IF (lCurrentTime.Value > (lToggleTime + lTogglePeriodMicroseconds)) THEN
	lToggle := NOT(lToggle);
	lToggleTime := lCurrentTime.Value;
END_IF

IF (lCurrentTime.Value > lIntegralClockTickPrevious) THEN
	lIntegralClockTick := TRUE;
	lIntegralClockTickPrevious := lIntegralClockTickPrevious + lIntegralPeriod;
ELSE
	lIntegralClockTick := FALSE;
END_IF

IF (lIntegralRunning) THEN
	lIntegralDuration := lCurrentTime.Value - lIntegralStartTime;
ELSE
	lIntegralStartTime := lCurrentTime.Value;
END_IF
IF (lIntegralReset) THEN
	lIntegralDuration := 0;
	lIntegralReset := FALSE;
END_IF

lCounter := lCounter + 1;


                
END_METHOD

METHOD initializeCycle
  VAR_INPUT
    currentTime : REFERENCE TO ULINT;
  END_VAR
                  lCurrentTime.InputReference REF= currentTime;

                
END_METHOD

METHOD describe
  VAR_INPUT
    executeContext : POINTER TO ExecuteContext;
  END_VAR
                  SUPER^.describe(executeContext);

IF (executeContext^.matchOption(cExecuteOptionSyntax)) THEN
	RETURN;
END_IF

IF (executeContext^.matchOption(cExecuteOptionParameter)) THEN	
	RETURN;
END_IF

executeContext^.appendPair('current_time',TIME_TO_STRING(ULINT_TO_TIME(lCurrentTime.Value/1000)),TRUE,TRUE);
executeContext^.appendPair('start_time',TIME_TO_STRING(ULINT_TO_TIME(lStartTime.Value/1000)),TRUE,TRUE);
executeContext^.appendPair('up_time',TIME_TO_STRING(ULINT_TO_TIME((lCurrentTime.Value - lStartTime.Value)/1000)),TRUE,TRUE);
executeContext^.appendPair('system_time',SystemTime,TRUE,TRUE);
executeContext^.appendPair('time_step',gTypeHandler.getTokenForUDINT(lTimeStep),FALSE,TRUE);

                
END_METHOD

METHOD configure
  VAR_INPUT
    executeContext : POINTER TO ExecuteContext;
  END_VAR
  VAR
    b : BOOL;
  END_VAR
                  IF (gSystemServices.Initialized) THEN
	IF (executeContext^.configureBool(cTokenFailSafeConfig,b,FALSE,0)) THEN
		RETURN;
	END_IF
END_IF

SUPER^.configure(executeContext);

                
END_METHOD

PROPERTY AverageCycleTime : ULINT
GET
                    AverageCycleTime := lAverageCycleTime;

                  
END_GET
END_PROPERTY

PROPERTY CycleTime : ULINT
GET
                    CycleTime := lCycleTime;

                  
END_GET
END_PROPERTY

PROPERTY Hours : REAL
GET
                    Hours := 0;
                  
END_GET
SET
                    
                  
END_SET
END_PROPERTY

PROPERTY IntegralClockTick : BOOL
GET
                    IntegralClockTick := lIntegralClockTick;
                  
END_GET
END_PROPERTY

PROPERTY OperationalHours : REAL
GET
                    OperationalHours := 0;
                  
END_GET
SET
                    
                  
END_SET
END_PROPERTY

PROPERTY SystemTime : REFERENCE TO t_medium_string
GET
                    SystemTime REF= lSystemTime;

                  
END_GET
END_PROPERTY

PROPERTY TimeStep : t_timestep
GET
                    TimeStep := lTimeStep;
                  
END_GET
END_PROPERTY

PROPERTY Toggle : BOOL
GET
                    Toggle := lToggle;
                  
END_GET
END_PROPERTY

PROPERTY TypeToken : t_medium_string
GET
                    TypeToken := 'Cycle';
                  
END_GET
END_PROPERTY

PROPERTY SystemTimeMicroseconds : ULINT
GET
                    SystemTimeMicroseconds := lCurrentTime.Value;
                  
END_GET
END_PROPERTY

PROPERTY StartCount : UINT
GET
                    StartCount := lStartCount.Value;
                  
END_GET
END_PROPERTY

PROPERTY StartTimeMicroseconds : ULINT
GET
                    StartTimeMicroseconds := 0; //lStartTime.Value;
                  
END_GET
END_PROPERTY
END_FUNCTION_BLOCK

FUNCTION_BLOCK Executor EXTENDS OperationalParticleSet
  VAR CONSTANT
    cCommandQueueMax : USINT := 4;
  END_VAR
  VAR
    lAlarmSoftwareCrash : ReportableAlarm;
    lClient : TCPClient;
    lExecuteContext : ExecuteContextExecutor;
    lExecuteContextParameterUpdate : ExecuteContextExecutor;
    lEnabled : BOOL := TRUE;
    lCommandQueue : ARRAY[1..cCommandQueueMax] OF t_command_request;
    lQueueCount : USINT := 0;
  END_VAR

            
          

METHOD operator
  VAR
    length : UINT;
  END_VAR
                  SUPER^.operator();

lExecuteContext.operator();
IF (lEnabled) THEN
	lClient.write(lExecuteContext.WriteStream^.Buffer,lExecuteContext.WriteStream^.Characters);
	lClient.write(lExecuteContextParameterUpdate.WriteStream^.Buffer,lExecuteContextParameterUpdate.WriteStream^.Characters);
END_IF

lExecuteContextParameterUpdate.WriteStream^.clear();

                
END_METHOD

METHOD initialize
                  lExecuteContext.Source REF= THIS^;
// lExecuteContextParameterUpdate.Source REF= THIS^; dummy executor: provides context only for direct write out

lAlarmSoftwareCrash.initializeState(NopSelf,'',cACExecutionFailed);

registerOperational(ADR(lClient));

SUPER^.initialize();

lExecuteContext.WriteStream^.IndentStr := '';
lExecuteContext.WriteStream^.NewlineStr := '$n';
lExecuteContext.WriteStream^.RecordInitiatorStr := '{';
lExecuteContext.WriteStream^.RecordTerminatorStr := '}';
lExecuteContext.WriteStream^.clear();
lExecuteContext.EnableExecutor := FALSE;

lExecuteContextParameterUpdate.WriteStream^.IndentStr := '';
lExecuteContextParameterUpdate.WriteStream^.NewlineStr := '$n';
lExecuteContextParameterUpdate.WriteStream^.RecordInitiatorStr := '{';
lExecuteContextParameterUpdate.WriteStream^.RecordTerminatorStr := '}';
lExecuteContextParameterUpdate.WriteStream^.clear();
lExecuteContextParameterUpdate.Command.optionCount := 1;
lExecuteContextParameterUpdate.Command.options[1] := cExecuteOptionParameter;
lExecuteContextParameterUpdate.EnableExecutor := FALSE;

                
END_METHOD

METHOD getNextExecuteCommand : BOOL
  VAR_INPUT
    command : REFERENCE TO t_command_request;
  END_VAR
  VAR
    i : USINT;
  END_VAR
                  IF (lQueueCount=0) THEN
	getNextExecuteCommand := FALSE;
	RETURN;
END_IF

command := lCommandQueue[1];

FOR i:=1 TO lQueueCount-1 DO
	lCommandQueue[i] := lCommandQueue[i+1];
END_FOR

lQueueCount := lQueueCount - 1;

getNextExecuteCommand := TRUE;

                
END_METHOD

METHOD reportParameterUpdates
  VAR_INPUT
    particle : POINTER TO t_particle;
  END_VAR
                  IF (particle=0) THEN
	RETURN;
END_IF

particle^.describe(ADR(lExecuteContextParameterUpdate));

                
END_METHOD

METHOD putCommand : BOOL
  VAR_INPUT
    command : REFERENCE TO t_command_request;
  END_VAR
                  IF (lQueueCount=cCommandQueueMax) THEN
	putCommand := FALSE;
	RETURN;
END_IF

lQueueCount := lQueueCount + 1;
lCommandQueue[lQueueCount] := command;

putCommand := TRUE;

                
END_METHOD

PROPERTY Client : REFERENCE TO TCPClient
GET
                    Client ref= lClient;
                  
END_GET
END_PROPERTY

PROPERTY TypeToken : t_medium_string
GET
                    TypeToken := 'Executor';
                  
END_GET
END_PROPERTY

PROPERTY ExecuteContext : POINTER TO ExecuteContextExecutor
GET
                    ExecuteContext:= ADR(lExecuteContext);
                  
END_GET
END_PROPERTY
END_FUNCTION_BLOCK

FUNCTION fCheckChannelMask : BOOL
  VAR_INPUT
    set : UINT;
    mask : t_channel_mask;
  END_VAR

            fCheckChannelMask := UINT_TO_BOOL(set AND INT_TO_UINT(mask));

          
END_FUNCTION

FUNCTION fCheckDebugFlags : BOOL
  VAR_INPUT
    mask : t_debug_mask;
  END_VAR

            fCheckDebugFlags := UINT_TO_BOOL(gDebugFlags.Value AND INT_TO_UINT(mask));

          
END_FUNCTION

FUNCTION_BLOCK LEDDiagnostic EXTENDS OperationalParticleSet
  VAR
    lCode : t_led_code;
  END_VAR

            
          

METHOD initialize
                  SUPER^.initialize();
SubSystem := cSubsystemPowerpack;

                
END_METHOD

METHOD operator
  VAR
    i : USINT;
  END_VAR
                  SUPER^.operator();

lCode := cLEDCodeNone;

                
END_METHOD

METHOD configure
  VAR_INPUT
    executeContext : POINTER TO ExecuteContext;
  END_VAR
  VAR
    b : BOOL;
  END_VAR
                  IF (gSystemServices.Initialized) THEN
	IF (executeContext^.configureBool(cTokenFailSafeConfig,b,FALSE,0)) THEN
		RETURN;
	END_IF
END_IF

SUPER^.configure(executeContext);

                
END_METHOD

PROPERTY TypeToken : t_medium_string
GET
                    TypeToken := 'LED';
                  
END_GET
END_PROPERTY

PROPERTY Code : t_led_code
GET
                    Code := lCode;
                  
END_GET
SET
                    // exceptions to the order rule
lCode := MAX(Code,lCode);

                  
END_SET
END_PROPERTY
END_FUNCTION_BLOCK

FUNCTION_BLOCK LocalMachine EXTENDS NonOperationalParticleSet
  VAR CONSTANT
    cRecoveryDetectionSteps : USINT := 3;
    cRecoverDetectionInterval : t_time := TIME#1s0ms;
  END_VAR
  VAR
    lVRMachineName : ValueReferencePersistentMediumString;
    lMachineName : t_persistent_medium_string;
    lVRDebugFlags : ValueReferencePersistentUINT;
    lVRFailSafeDebugFlags : ValueReferencePersistentUINT;
    lFailSafeDebugFlags : t_persistent_uint;
    lRecoveryDetectionStep : t_persistent_uint;
    lRecoveryDetectionStepActive : t_persistent_bool;
    lRecoveryDetectionPeriods : ARRAY[0..cRecoveryDetectionSteps] OF t_time;
    lRecoveryDetectionTimerLower : t_timer;
    lRecoveryDetectionTimerUpper : t_timer;
    lRecoveryDetectionSuccess : BOOL := FALSE;
    lPostInitialize : BOOL := TRUE;
  END_VAR

            
          

METHOD execute
  VAR_INPUT
    executeContext : POINTER TO ExecuteContext;
  END_VAR
  VAR
    token : t_token_string;
    mask : t_debug_mask;
  END_VAR
                  IF (executeContext=0) THEN
	RETURN;
END_IF

IF (executeContext^.matchCommand(sCommandDebugMaskAdd)) THEN

	IF (NOT(executeContext^.configureEnum(cEnumTypeDebugMask,cTokenFeature,mask,TRUE,THIS))) THEN
		RETURN;
	END_IF
	
	gDebugFlags.Value := gDebugFlags.Value OR INT_TO_UINT(mask);
	RETURN;
END_IF

IF (executeContext^.matchCommand(sCommandDebugMaskDelete)) THEN

	IF (NOT(executeContext^.configureEnum(cEnumTypeDebugMask,cTokenFeature,mask,TRUE,THIS))) THEN
		RETURN;
	END_IF
	
	gDebugFlags.Value := gDebugFlags.Value AND NOT(INT_TO_UINT(mask));
	RETURN;
END_IF

IF (executeContext^.matchCommand(sCommandDebugMaskClear)) THEN	
	gDebugFlags.Value := 0;
	RETURN;
END_IF

SUPER^.execute(executeContext);

                
END_METHOD

METHOD postInitialize
                  lPostInitialize := false;
                
END_METHOD

METHOD initialize
                  lVRDebugFlags.initializeValueReference(gDebugFlags,NopSelf,'Debug','System wide debug flags','',cValueStyleParameter);

lVRFailSafeDebugFlags.initializeValueReference(lFailSafeDebugFlags,NopSelf,'FailSafeDebug','Failsafe debug flags','',cValueStyleParameter);
lFailSafeDebugFlags.Identifier := t_persistent_id.cPersistentID_FailSafeDebugFlags;
lFailSafeDebugFlags.initialize();

lVRMachineName.initializeValueReference(lMachineName,NopSelf,'MachineName','Name of the machine','',cValueStyleParameter);
lMachineName.Identifier := t_persistent_id.cPersistentID_MachineName;
lMachineName.initialize();

lRecoveryDetectionStep.Identifier := t_persistent_id.cPersistentID_RecoveryDetectionStep;
lRecoveryDetectionStep.initialize();

lRecoveryDetectionStepActive.Identifier := t_persistent_id.cPersistentID_RecoveryDetectionStepActive;
lRecoveryDetectionStepActive.initialize();

SUPER^.initialize();
SubSystem := cSubsystemMachine;

lRecoveryDetectionPeriods[0] := T#500MS;
lRecoveryDetectionPeriods[1] := T#2500MS;
lRecoveryDetectionPeriods[2] := T#500MS;
lRecoveryDetectionPeriods[3] := T#2500MS;

lRecoveryDetectionTimerLower.Enable := TRUE;
lRecoveryDetectionTimerLower.Period := lRecoveryDetectionPeriods[MIN(lRecoveryDetectionStep.Value,cRecoveryDetectionSteps)];
lRecoveryDetectionTimerLower.initialize();

lRecoveryDetectionTimerUpper.Enable := TRUE;
lRecoveryDetectionTimerUpper.Period := lRecoveryDetectionPeriods[MIN(lRecoveryDetectionStep.Value,cRecoveryDetectionSteps)] + cRecoverDetectionInterval;
lRecoveryDetectionTimerUpper.initialize();

IF (lRecoveryDetectionStepActive.Value) THEN
	lRecoveryDetectionStep.Value := lRecoveryDetectionStep.Value + 1;
	lRecoveryDetectionStepActive.Value := FALSE;
END_IF

IF (lRecoveryDetectionStep.Value>cRecoveryDetectionSteps) THEN
	lRecoveryDetectionStep.Value := 0;
	lRecoveryDetectionSuccess := TRUE;
	gDebugFlags.Value := INT_TO_UINT(cDebugDisableWatchdog);
END_IF
                
END_METHOD

METHOD operator
                  SUPER^.operator();

IF (gSystemServices.PLC.CrashSeverity>3) THEN
	lFailSafeDebugFlags.Value := INT_TO_UINT(cDebugDisableWatchdog);
END_IF

IF (gSystemServices.PLC.CrashSeverity>2) THEN
	gDebugFlags.Value := lFailSafeDebugFlags.Value;
END_IF

IF (lRecoveryDetectionTimerUpper.Enable) THEN
	lRecoveryDetectionTimerLower.operator();
	lRecoveryDetectionTimerUpper.operator();

	lRecoveryDetectionStepActive.Value := ((lRecoveryDetectionTimerLower.Expired) AND
		(NOT(lRecoveryDetectionTimerUpper.Expired)));

	IF ((lRecoveryDetectionTimerLower.Expired) AND
		(lRecoveryDetectionTimerUpper.Expired)) THEN
		lRecoveryDetectionTimerLower.Enable := FALSE;
		lRecoveryDetectionTimerUpper.Enable := FALSE;
		lRecoveryDetectionStep.Value := 0;
	END_IF
END_IF

IF (lPostInitialize) THEN
	postInitialize();
END_IF

                
END_METHOD

METHOD defaultPersistence
                  lFailSafeDebugFlags.Value := INT_TO_UINT(cDebugDisableWatchdog);
                
END_METHOD

METHOD describe
  VAR_INPUT
    executeContext : POINTER TO ExecuteContext;
  END_VAR
                  SUPER^.describe(executeContext);

IF (executeContext^.matchOption(cExecuteOptionSyntax)) THEN
	executeContext^.describeSyntaxExecutable(sCommandDebugMaskAdd);
	executeContext^.describeSyntaxExecutable(sCommandDebugMaskDelete);
	executeContext^.describeSyntaxExecutable(sCommandDebugMaskClear);

	RETURN;
END_IF

IF (executeContext^.matchOption(cExecuteOptionParameter)) THEN	
	RETURN;
END_IF

executeContext^.appendPair('machine_name',lMachineName.Value,TRUE,TRUE);


                
END_METHOD

METHOD configure
  VAR_INPUT
    executeContext : POINTER TO ExecuteContext;
  END_VAR
  VAR
    b : BOOL;
  END_VAR
                  IF (gSystemServices.Initialized) THEN
	IF (executeContext^.configureBool(cTokenFailSafeConfig,b,FALSE,0)) THEN
		RETURN;
	END_IF
END_IF

SUPER^.configure(executeContext);

                
END_METHOD

PROPERTY MachineName : t_medium_string
GET
                    MachineName := lMachineName.Value;
                  
END_GET
SET
                    lMachineName.Value := MachineName;
                  
END_SET
END_PROPERTY

PROPERTY TypeToken : t_medium_string
GET
                    TypeToken := 'Local';
                  
END_GET
END_PROPERTY
END_FUNCTION_BLOCK

FUNCTION_BLOCK Peripheral EXTENDS OperationalParticleSet
  VAR
    lExternalState : REFERENCE TO UINT;
    lSupplementaryCommand : REFERENCE TO USINT;
    lInternalState : REFERENCE TO USINT;
    lReportableState : REFERENCE TO UDINT;
    lSupplementaryState : REFERENCE TO UINT;
    lOperatingModeLockRequest : ValueObjectBoolInputReferenceUSINT;
    lOperatingModeRunningRegister : ValueObjectBoolInputReferenceUSINT;
    lUMFSRegister : ValueObjectBoolInputReferenceUSINT;
    lValidTransmissions : ValueObjectBoolInputReferenceUSINT;
    lTPDO1Stuffing : ValueObjectBoolInputReferenceUSINT;
    lReportable : ARRAY[0..31] OF POINTER TO t_reportable;
  END_VAR

            ;
          

METHOD initialize
                  IF ((NOT(__ISVALIDREF(lExternalState))) OR
	(NOT(__ISVALIDREF(lSupplementaryCommand))) OR
	(NOT(__ISVALIDREF(lInternalState))) OR
	(NOT(__ISVALIDREF(lReportableState))) OR
	(NOT(__ISVALIDREF(lSupplementaryState)))) THEN
	gCodeErrorHandler(pMessage:=CONCAT('null reference in ',lIdentity));
END_IF

lOperatingModeLockRequest.initializeValueObjectOp(OpSelf,'LockReq','Lock operating mode requested','',cValueStyleConfigurable);
lOperatingModeLockRequest.Index := 0;
lOperatingModeLockRequest.InputReference REF= lInternalState;

lOperatingModeRunningRegister.initializeValueObjectOp(OpSelf,'RunningReg','Running operating mode requested','',cValueStyleConfigurable);
lOperatingModeRunningRegister.Index := 1;
lOperatingModeRunningRegister.InputReference REF= lInternalState;

lUMFSRegister.initializeValueObjectOp(OpSelf,'UMFSReg','UMFS registration requested','',cValueStyleConfigurable);
lUMFSRegister.Index := 2;
lUMFSRegister.InputReference REF= lInternalState;

lValidTransmissions.initializeValueObjectOp(OpSelf,'ValidTrnsmssns','Valid transmissions detected','',cValueStyleConfigurable);
lValidTransmissions.Index := 3;
lValidTransmissions.InputReference REF= lInternalState;

lTPDO1Stuffing.initializeValueObjectOp(OpSelf,'TPDO1Stuffing','TPDO1 stuffing bit detected','',cValueStyleConfigurable);
lTPDO1Stuffing.Index := 7;
lTPDO1Stuffing.InputReference REF= lInternalState;

SUPER^.initialize();
                
END_METHOD

METHOD initializePeripheral
  VAR_INPUT
    externalState : REFERENCE TO UINT;
    supplementaryCommand : REFERENCE TO USINT;
    internalState : REFERENCE TO USINT;
    reportableState : REFERENCE TO UDINT;
    supplementaryState : REFERENCE TO UINT;
  END_VAR
                  lExternalState REF= externalState;
lSupplementaryCommand REF= supplementaryCommand;

lInternalState REF= internalState;
lReportableState REF= reportableState;
lSupplementaryState REF= supplementaryState;



                
END_METHOD

METHOD operator
  VAR
    i : USINT;
    u : UDINT;
  END_VAR
                  SUPER^.operator();

(* traffic FROM master PLC *)

lExternalState := 0;
lExternalState := fMergeBoolIntoWord(pWord:=lExternalState,pData:=gManualTemporaryOveride,pStart:=9);

(* traffic to master PLC *)

u := lReportableState;
FOR i:=0 TO 15 DO
	IF ((UDINT_TO_BOOL(u AND 2#1)) AND
		(lReportable[i]<>0)) THEN
		lReportable[i]^.trigger(FALSE);
	END_IF
	
	u := SHR(u,1);
END_FOR

                
END_METHOD

METHOD registerReportable
  VAR_INPUT
    reportable : POINTER TO t_reportable;
    index : USINT;
  END_VAR
                  IF (index>31) THEN
	RETURN;
END_IF

lReportable[index] := reportable;

                
END_METHOD

PROPERTY TPDO1Stuffing : BOOL
GET
                    TPDO1Stuffing := lTPDO1Stuffing.Value;
                  
END_GET
END_PROPERTY

PROPERTY TypeToken : t_medium_string
GET
                    TypeToken := 'Peripheral';
                  
END_GET
END_PROPERTY

PROPERTY ValidTransmissions : BOOL
GET
                    ValidTransmissions := lValidTransmissions.Value;
                  
END_GET
END_PROPERTY

PROPERTY SupplementaryCommand : REFERENCE TO USINT
GET
                    SupplementaryCommand ref= lSupplementaryCommand;
                  
END_GET
END_PROPERTY

PROPERTY SupplementaryState : REFERENCE TO UINT
GET
                    SupplementaryState ref= lSupplementaryState;
                  
END_GET
END_PROPERTY
END_FUNCTION_BLOCK

FUNCTION_BLOCK PLC EXTENDS OperationalParticleSet
  VAR CONSTANT
    cCrashDetectionPeriod : t_time := TIME#30s0ms;
    cPersistedCommandCount : USINT := 100;
  END_VAR
  VAR
    lVRTriggerWipePersistence : ValueReferenceBool;
    lTriggerWipePersistence : BOOL := FALSE;
    lVRTriggerDefaultPersistence : ValueReferenceBool;
    lTriggerDefaultPersistence : BOOL := FALSE;
    lVRTriggerResetSoftwareCrashCount : ValueReferenceBool;
    lTriggerResetSoftwareCrashCount : BOOL := FALSE;
    lVRTemporaryDisableWatchdog : ValueReferencePersistentBool;
    lTemporaryDisableWatchdog : t_persistent_bool;
    lVRMaintenanceMode : ValueReferenceBool;
    lMaintenanceMode : BOOL := FALSE;
    lMaintenanceModePrevious : BOOL := FALSE;
    lAlarmSoftwareCrash : ReportableAlarm;
    lAlarmFailSafeMode : ReportableAlarm;
    lAlarmMaintenanceMode : ReportableAlarm;
    lAlarmWatchdogDisabled : ReportableAlarm;
    lAlarmPersistedCommands : ReportableAlarm;
    lShutdownCode : t_persistent_int;
    lPreviousShutdownCode : t_shutdown_code;
    lSoftwareCrashCount : t_persistent_uint;
    lCrashSeverity : t_persistent_uint;
    lCrashDetectionTimer : t_timer;
    lCrashDetected : BOOL := FALSE;
    lTrapDetected : BOOL := FALSE;
    lFailSafeModeActive : BOOL := FALSE;
    lDisableWatchDog : BOOL := FALSE;
    lForceDisableWatchDog : BOOL := FALSE;
    lPersistedCommands : ARRAY[1..cPersistedCommandCount] OF PersistentCommand;
    lPersistedCommandCount : UINT;
    lPersistedCommandsStatus : BOOL := TRUE;
  END_VAR

            
          

METHOD setFailSafeMode
                  lFailSafeModeActive := TRUE;

setWatchdog();


                
END_METHOD

METHOD clearFailSafeMode
                  lFailSafeModeActive := FALSE;

setWatchdog();

                
END_METHOD

METHOD operator
  VAR
    i : USINT;
  END_VAR
                  SUPER^.operator();

IF (lTriggerWipePersistence) THEN
	lTriggerWipePersistence := FALSE;

	gPersistenceManager.clear();

	defaultPersistence();
	gSystemServices.LocalMachine.defaultPersistence();
END_IF

IF (lTriggerDefaultPersistence) THEN
	lTriggerDefaultPersistence := FALSE;

	defaultPersistence();
	gSystemServices.LocalMachine.defaultPersistence();
END_IF
	
IF (lTriggerResetSoftwareCrashCount) THEN
	lTriggerResetSoftwareCrashCount := FALSE;

	lSoftwareCrashCount.Value := 0;
END_IF

IF (lCrashDetectionTimer.Enable) THEN
	lCrashDetectionTimer.operator();
	IF (lCrashDetectionTimer.Expired) THEN
		lCrashDetectionTimer.Enable := FALSE;
		lShutdownCode.Value := t_shutdown_code.cShutdownCodeUnknown;
	END_IF
END_IF

IF ((lCrashDetected) OR (lTrapDetected)) THEN
	lAlarmSoftwareCrash.trigger(FALSE);
	gSystemServices.LEDDiagnostic.Code := cLEDCodeSoftwareCrash;
END_IF

IF (lFailSafeModeActive) THEN
	lAlarmFailSafeMode.trigger(FALSE);

	IF (lCrashSeverity.Value>1) THEN
		gSystemServices.LEDDiagnostic.Code := cLEDCodeFailSafeSevere;			
	ELSE
		gSystemServices.LEDDiagnostic.Code := cLEDCodeFailSafe;
	END_IF
END_IF

IF (MaintenanceMode<>lMaintenanceModePrevious) THEN
	lMaintenanceModePrevious := MaintenanceMode;
	setWatchdog();	
END_IF

IF (MaintenanceMode)  THEN
	lAlarmMaintenanceMode.trigger(FALSE);
	gSystemServices.LEDDiagnostic.Code := cLEDCodeMaintenance;
END_IF

IF (fCheckDebugFlags(cDebugDisableWatchdog)<>lDisableWatchDog) THEN
	lDisableWatchDog := NOT(lDisableWatchDog);
	setWatchdog();
END_IF

IF ((lDisableWatchDog) OR (lForceDisableWatchDog)) THEN
	lAlarmWatchdogDisabled.trigger(FALSE);
	gSystemServices.LEDDiagnostic.Code := cLEDCodeWatchDogDisabled;	
END_IF

IF (NOT(lPersistedCommandsStatus)) THEN
	lAlarmPersistedCommands.trigger(FALSE);
END_IF

                
END_METHOD

METHOD initialize
  VAR
    i : USINT;
    id : INT;
  END_VAR
                  lVRTriggerWipePersistence.initializeValueReference(lTriggerWipePersistence,NopSelf,'WipePersist','Trigger wipe of persistent memory','',cValueStyleTrigger);
lVRTriggerDefaultPersistence.initializeValueReference(lTriggerDefaultPersistence,NopSelf,'DefaultPersist','Trigger loading default persistent memory','',cValueStyleTrigger);
lVRTriggerResetSoftwareCrashCount.initializeValueReference(lTriggerResetSoftwareCrashCount,NopSelf,'ResetOpSwCrshCnt','Trigger reset software crash count','',cValueStyleTrigger);
lVRMaintenanceMode.initializeValueReference(lMaintenanceMode,NopSelf,'Maintenance','Whether in maintenance mode','',cValueStyleParameter);

lVRTemporaryDisableWatchdog.initializeValueReference(lTemporaryDisableWatchdog,NopSelf,'TmpDsblWatchDog','Temporarily disable watchdog','',cValueStyleParameter);
lTemporaryDisableWatchdog.Identifier := t_persistent_id.cPersistentID_TemporaryDisableWatchdog;
lTemporaryDisableWatchdog.initialize();

lAlarmSoftwareCrash.initializeState(NopSelf,'',cACSoftwareCrash);
lAlarmFailSafeMode.initializeState(NopSelf,'',cACFailSafeMode);
lAlarmMaintenanceMode.initializeState(NopSelf,'',cACMaintenanceMode);
lAlarmWatchdogDisabled.initializeState(NopSelf,'',cACWatchdogDisabled);
lAlarmPersistedCommands.initializeState(NopSelf,'',cACPersistedCommands);

lShutdownCode.Identifier := t_persistent_id.cPersistentID_ShutdownCode;
lShutdownCode.initialize();

lSoftwareCrashCount.Identifier := t_persistent_id.cPersistentID_SoftwareCrashCount;
lSoftwareCrashCount.initialize();

lCrashSeverity.Identifier := t_persistent_id.cPersistentID_CrashSeverity;
lCrashSeverity.initialize();

lDisableWatchDog := fCheckDebugFlags(cDebugDisableWatchdog);

IF (lTemporaryDisableWatchdog.Value) THEN
	lTemporaryDisableWatchdog.Value := FALSE;	
	lForceDisableWatchDog := TRUE;
END_IF

lPersistedCommandCount := 0;
id := t_persistent_id.cPersistentID_CommandRepositoryLower;

FOR i:=1 TO cPersistedCommandCount DO
	lPersistedCommands[i].Identifier := id;
	lPersistedCommands[i].initialize();
	
	id := id + UINT_TO_INT(lPersistedCommands[i].Blocks);
	
	IF (lPersistedCommands[i].Valid) THEN
		lPersistedCommandCount := lPersistedCommandCount + 1;
	END_IF
END_FOR
	
SUPER^.initialize();

lPreviousShutdownCode := lShutdownCode.Value;
lShutdownCode.Value := t_shutdown_code.cShutdownCodeCrashDetected;

lCrashDetected := (lPreviousShutdownCode=t_shutdown_code.cShutdownCodeCrashDetected);
IF (lCrashDetected) THEN		
	lCrashSeverity.Value := lCrashSeverity.Value + 1;
	lSoftwareCrashCount.Value := lSoftwareCrashCount.Value + 1;
ELSE
	lCrashSeverity.Value := 0;
END_IF

lCrashDetectionTimer.Enable := TRUE;
lCrashDetectionTimer.Period := cCrashDetectionPeriod;
lCrashDetectionTimer.initialize();

                
END_METHOD

METHOD describe
  VAR_INPUT
    executeContext : POINTER TO ExecuteContext;
  END_VAR
  VAR
    i : UINT;
    str : STRING;
    store : t_command_store;
    particle : t_particle_ptr;
    token : t_token_string;
  END_VAR
                  SUPER^.describe(executeContext);

IF (executeContext^.matchOption(cExecuteOptionSyntax)) THEN
	executeContext^.describeSyntaxExecutable(sCommandExport);
	executeContext^.describeSyntaxExecutable(sCommandClear);
	executeContext^.describeSyntaxExecutable(sCommandExecute);

	RETURN;
END_IF

IF (executeContext^.matchOption(cExecuteOptionParameter)) THEN	
	RETURN;
END_IF

executeContext^.appendPair('failsafe_active',gTypeHandler.getTokenForBool(lFailSafeModeActive),FALSE,TRUE);
executeContext^.appendPair('crash_detected',gTypeHandler.getTokenForBool(lCrashDetected),FALSE,TRUE);
executeContext^.appendPair('crash_severity',gTypeHandler.getTokenForUINT(lCrashSeverity.Value),FALSE,TRUE);
executeContext^.appendPair('previous_shutdown',gTypeHandler.getTokenForEnum(cEnumTypeShutdownCode,lPreviousShutdownCode),TRUE,TRUE);
executeContext^.appendPair('watchdog',gTypeHandler.getTokenForBool(NOT((lDisableWatchdog) OR (lForceDisableWatchDog))),FALSE,TRUE);
executeContext^.appendPair('persisted_count',gTypeHandler.getTokenForUINT(lPersistedCommandCount),FALSE,TRUE);
executeContext^.appendPair('persisted_status',gTypeHandler.getTokenForBool(lPersistedCommandsStatus),FALSE,TRUE);

IF (NOT(executeContext^.matchOption(cExecuteOptionVerbose))) THEN
	RETURN;
END_IF

executeContext^.append(', ');
executeContext^.WriteStream^.increaseIndent();
executeContext^.formatWithNewlineIndent();
executeContext^.append('"persisted": [');
executeContext^.WriteStream^.increaseIndent();

FOR i:=1 TO lPersistedCommandCount DO
	IF (NOT(lPersistedCommands[i].Valid)) THEN
		CONTINUE;
	END_IF
	
	executeContext^.recordInitiatorWithNewlineIndent();
	executeContext^.appendPair('index',gTypeHandler.getTokenForUINT(i),FALSE,FALSE);

	store := lPersistedCommands[i].Value;
	
	particle := gSystemServices.getParticle(token,store.particle);
	IF (particle=0) THEN
		CONTINUE;
	END_IF
	 
	str := particle^.lIdentity;
	str := CONCAT(str,' ');
	str := CONCAT(str,gTypeHandler.getTokenForEnum(cEnumTypeTokenType,store.command));
	
	FOR i:=1 TO store.optionCount DO
		str := CONCAT(str,' -');
		str := CONCAT(str,gTypeHandler.getTokenForEnum(cEnumTypeExecuteOption,store.options[i]));
	END_FOR
	
	FOR i:=1 TO store.argumentCount DO
		str := CONCAT(str,' ');
		str := CONCAT(str,gTypeHandler.getTokenForEnum(cEnumTypeTokenType,store.arguments[i].parameter));
		str := CONCAT(str,'=');
		str := CONCAT(str,store.arguments[i].value);
	END_FOR
	
	executeContext^.appendPair('command',str,TRUE,TRUE);
	executeContext^.recordTerminator();
	
	IF (i<lPersistedCommandCount) THEN
		executeContext^.append(', ');		
	END_IF
END_FOR

executeContext^.WriteStream^.decreaseIndent();
executeContext^.append(']');
executeContext^.WriteStream^.decreaseIndent();

                
END_METHOD

METHOD configure
  VAR_INPUT
    executeContext : POINTER TO ExecuteContext;
  END_VAR
  VAR
    index : UDINT := 0;
    data : UDINT := 0;
    b : BOOL;
  END_VAR
                  IF (gSystemServices.Initialized) THEN
	IF (executeContext^.configureBool(cTokenFailSafeConfig,b,FALSE,0)) THEN
		RETURN;
	END_IF
END_IF

(* eolus
IF (executeContext^.configureX(cTokenRawIndex)) THEN
	index := executeContext^.ParameterAsIndexToken;

	IF (index>gPersistenceManager.IndexMax) THEN
		executeContextFail(executeContext,cExecuteReturnIllegalIndex,TRUE);
		RETURN;
	END_IF
	
	data := executeContext^.configureUDINT(data);
	IF (NOT(executeContext^.Error)) THEN
		gPersistenceManager.write(index,UDINT_TO_DWORD(data));
	END_IF

	RETURN;
END_IF*)

SUPER^.configure(executeContext);

                
END_METHOD

METHOD setWatchdogDebug
                  
                
END_METHOD

METHOD setWatchdogNormal
                  
                
END_METHOD

METHOD setWatchdog
                  IF ((lDisableWatchdog) OR (lForceDisableWatchDog)) THEN
	setWatchdogDisabled();
	RETURN;
END_IF

IF ((MaintenanceMode) OR
	(FailSafeModeActive) OR
	(NOT(gSystemServices.Initialized))) THEN
	setWatchdogDebug();
	RETURN;
END_IF

setWatchdogNormal();	

                
END_METHOD

METHOD setWatchdogDisabled
                  
                
END_METHOD

METHOD execute
  VAR_INPUT
    executeContext : POINTER TO ExecuteContext;
  END_VAR
  VAR
    udi : UDINT;
    i : UINT;
    comma : BOOL;
    index : UINT;
  END_VAR
                  IF (executeContext^.matchCommand(sCommandExport)) THEN

	executeContext^.recordInitiator();
	executeContext^.appendPair('identity',lIdentity,TRUE,FALSE);
	executeContext^.append(',"persistent-memory": [');

	comma := FALSE;
	FOR udi:=0 TO gPersistenceManager.IndexMax DO
		executeContext^.appendPair(UDINT_TO_STRING(i),gTypeHandler.getTokenForUDINT(DWORD_TO_UDINT(gPersistenceManager.read(udi))),FALSE,comma);
		comma := TRUE;
	END_FOR
	
	executeContext^.append(']');
	executeContext^.recordTerminatorWithNewline();

	RETURN;
END_IF

IF (executeContext^.matchCommand(sCommandClear)) THEN
	IF (executeContext^.matchOption(cExecuteOptionAll)) THEN
		FOR i:=1 TO cPersistedCommandCount DO
			clearCommand(i);
		END_FOR

		RETURN;
	END_IF

	IF (NOT(executeContext^.configureUINT(cTokenIndex,index,TRUE,0))) THEN
		RETURN;
	END_IF

	IF (index>cPersistedCommandCount) THEN
		executeContextFail(THIS,cExecuteReturnIllegalIndex,TRUE);
		RETURN;
	END_IF
	
	clearCommand(index);

	RETURN;
END_IF

IF (executeContext^.matchCommand(sCommandExecute)) THEN
	IF (executeContext^.matchOption(cExecuteOptionAll)) THEN
		executeAllCommands();

		RETURN;
	END_IF

	IF (NOT(executeContext^.configureUINT(cTokenIndex,index,TRUE,0))) THEN
		RETURN;
	END_IF

	IF (index>cPersistedCommandCount) THEN
		executeContextFail(THIS,cExecuteReturnIllegalIndex,TRUE);
		RETURN;
	END_IF
	
	executeCommand(index);

	RETURN;
END_IF

SUPER^.execute(executeContext);

                
END_METHOD

METHOD defaultPersistence
  VAR
    i : UINT;
  END_VAR
                  FOR i:=1 TO cPersistedCommandCount DO
	clearCommand(i);
END_FOR

                
END_METHOD

METHOD executeCommand : BOOL
  VAR_INPUT
    index : UINT;
  END_VAR
  VAR
    store : t_command_store;
    command : t_command_request;
    token : t_token_string;
  END_VAR
                  executeCommand := FALSE;

IF (index>cPersistedCommandCount) THEN
	RETURN;
END_IF

store := lPersistedCommands[index].Value;

command.particle := gSystemServices.getParticle(token,store.particle);
IF (command.particle=0) THEN
	RETURN;
END_IF

command.command := store.command;
command.argumentCount := store.argumentCount;
command.arguments := store.arguments;
command.optionCount := store.optionCount;
command.options := store.options;

executeCommand := gSystemServices.Executor.putCommand(command);

                
END_METHOD

METHOD executeAllCommands : BOOL
  VAR
    i : UINT;
  END_VAR
                  lPersistedCommandsStatus := TRUE;

FOR i:=1 TO cPersistedCommandCount DO
	IF (NOT(executeCommand(i))) THEN
		lPersistedCommandsStatus := FALSE;
	END_IF
END_FOR

executeAllCommands := lPersistedCommandsStatus;

                
END_METHOD

METHOD persistCommand : BOOL
  VAR_INPUT
    command : REFERENCE TO t_command_request;
  END_VAR
  VAR
    store : t_command_store;
    i : UINT;
    j : UINT;
  END_VAR
                  IF ((command.particle=0) OR
	(lPersistedCommandCount=cPersistedCommandCount)) THEN
	persistCommand := FALSE;
	RETURN;
END_IF

store.particle := command.particle^.lParticleId;

store.argumentCount := command.argumentCount;
store.arguments := command.arguments;
store.command := command.command;
store.optionCount := command.optionCount;
store.options := command.options;

FOR i:=1 TO store.optionCount DO
	IF (store.options[i]=cExecuteOptionPersist) THEN		
		store.optionCount := store.optionCount - 1;
		FOR j:=i TO store.optionCount DO
			store.options[j] := store.options[j+1];
		END_FOR	
	END_IF
END_FOR

FOR i:=1 TO cPersistedCommandCount DO
	IF (NOT(lPersistedCommands[i].Valid)) THEN
		lPersistedCommands[i].Value := store;
		lPersistedCommandCount := lPersistedCommandCount + 1;

		persistCommand := TRUE;
		RETURN;
	END_IF
END_FOR

persistCommand := FALSE;


                
END_METHOD

METHOD clearCommand
  VAR_INPUT
    index : UINT;
  END_VAR
  VAR
    store : t_command_store;
  END_VAR
                  IF (index>cPersistedCommandCount) THEN
	RETURN;
END_IF

store.particle := 0;
store.command := 0;
store.optionCount := 0;
store.argumentCount := 0;

IF ((lPersistedCommands[index].Valid) AND
	(lPersistedCommandCount>0)) THEN
	lPersistedCommandCount := lPersistedCommandCount - 1;
END_IF

lPersistedCommands[index].Value := store;

                
END_METHOD

PROPERTY TrapDetected : BOOL
GET
                    TrapDetected := lTrapDetected;
                  
END_GET
END_PROPERTY

PROPERTY PreviousShutdownCode : t_shutdown_code
GET
                    PreviousShutdownCode := lPreviousShutdownCode;
                  
END_GET
END_PROPERTY

PROPERTY SoftwareCrashCount : UINT
GET
                    SoftwareCrashCount := lSoftwareCrashCount.Value;
                  
END_GET
END_PROPERTY

PROPERTY CrashDetected : BOOL
GET
                    CrashDetected := lCrashDetected;
                  
END_GET
END_PROPERTY

PROPERTY TypeToken : t_medium_string
GET
                    TypeToken := 'PLC';
                  
END_GET
END_PROPERTY

PROPERTY CrashSeverity : UINT
GET
                    
                  
END_GET
END_PROPERTY

PROPERTY FailSafeModeActive : BOOL
GET
                    FailSafeModeActive := lFailSafeModeActive;
                  
END_GET
END_PROPERTY

PROPERTY MaintenanceMode : BOOL
GET
                    MaintenanceMode := lMaintenanceMode;
                  
END_GET
END_PROPERTY
END_FUNCTION_BLOCK

FUNCTION_BLOCK SubSystemState EXTENDS SystemState
  VAR
    lCausalSyncState : ReportableCausal;
    lMasterSystemState : ValueObjectEnumType;
    lLowerSyncState : t_system_state := cSystemStatePreOperational;
    lUpperSyncState : t_system_state := cSystemStateOperational;
  END_VAR

            ;
          

METHOD initialize
                  lCausalSyncState.initializeState(NopSelf,'',cCCSyncState);

lMasterSystemState.EnumType := cEnumTypeSystemState;
lMasterSystemState.initializeValueObject(NopSelf,'Master','System state of master','',cValueStyleConfigurable);

SUPER^.initialize();

lAutomaticStart := TRUE;



                
END_METHOD

METHOD operator
                  lMasterSystemState.operator();
IF ((lMasterSystemState.Value<=lLowerSyncState) OR
	(lMasterSystemState.Value>lUpperSyncState)) THEN
	transitionForceMax(lMasterSystemState.Value,ADR(lCausalSyncState),lCausalSyncState.Override);
END_IF

SUPER^.operator();


                
END_METHOD

PROPERTY LowerSyncState : t_system_state
GET
                    LowerSyncState := lLowerSyncState;
                  
END_GET
SET
                    lLowerSyncState := LowerSyncState;
                  
END_SET
END_PROPERTY

PROPERTY UpperSyncState : t_system_state
GET
                    UpperSyncState := lUpperSyncState;
                  
END_GET
SET
                    lUpperSyncState := UpperSyncState;
                  
END_SET
END_PROPERTY
END_FUNCTION_BLOCK

FUNCTION_BLOCK System EXTENDS OperationalParticleSet
  VAR CONSTANT
    cSubsystemSetMax : USINT := 64;
  END_VAR
  VAR
    lVRTriggerClearFailSafeMode : ValueReferenceBool;
    lTriggerClearFailSafeMode : BOOL;
    _LocalMachine : REFERENCE TO LocalMachine;
    _LEDDiagnostic : REFERENCE TO LEDDiagnostic;
    _ReportableChannelManager : REFERENCE TO ReportableChannelManager;
    _Executor : REFERENCE TO Executor;
    _Cycle : REFERENCE TO Cycle;
    _PLC : REFERENCE TO PLC;
    _SystemState : REFERENCE TO SystemState;
    lInitializationStage : SINT := -1;
    lInitialized : BOOL := FALSE;
    lSubsystemCount : USINT := 0;
    lSubsystemSet : ARRAY[1..cSubsystemSetMax] OF t_particle_ptr;
  END_VAR

            ;
          

METHOD parseString
  VAR_INPUT
    str : t_long_string;
  END_VAR
                  lReadStream.clear();
lReadStream.appendPtr(ADR(str));
lReadStream.initializeParsing();

lWriteStream.clear();
//eolus IF ((NOT(parse(ADR(lReadStream),ADR(lWriteStream),TRUE))) OR
//eolus 	(lReadStream.CurrentToken=cTokenError) OR 
//eolus 	(lReadStream.CurrentToken=cTokenOverflow)) THEN
//eolus 	gCodeErrorHandler(pMessage:='Syntax error - bad string');
//eolus END_IF

                
END_METHOD

METHOD recurse
  VAR_INPUT
    executeContext : POINTER TO ExecuteContext;
  END_VAR
  VAR
    i : USINT;
  END_VAR
                  SUPER^.recurse(executeContext);

IF (NOT(executeContext^.matchOption(cExecuteOptionSubsystems))) THEN	
	RETURN;
END_IF

FOR i:=1 TO lSubsystemCount DO
	lSubsystemSet[i]^.recurse(executeContext);
END_FOR

                
END_METHOD

METHOD initialize
  VAR
    i : USINT;
  END_VAR
                  lFeature := false;

SUPER^.initialize();

FOR i:=1 TO lSubsystemCount DO
	IF (lSubsystemSet[i]^.lParticleId=0) THEN
		lSubsystemSet[i]^.initialize();
	END_IF
END_FOR
                
END_METHOD

METHOD operator
  VAR
    i : USINT;
  END_VAR
                  IF (lTriggerClearFailSafeMode) THEN
	lTriggerClearFailSafeMode := FALSE;
	clearFailSafeMode();
END_IF

IF (lInitializationStage<1) THEN
	RETURN;
END_IF

FOR i:=1 TO lSubsystemCount DO
	IF (lSubsystemSet[i]^.lProceed) THEN
		lSubsystemSet[i]^.operator();
	END_IF
END_FOR

SUPER^.operator();

IF (NOT(lInitialized)) THEN
	gSystemServices.LEDDiagnostic.Code := cLEDCodeStartup;
END_IF
                
END_METHOD

METHOD clearFailSafeMode
                  FailSafeMode := FALSE;

gSystemServices.PLC.clearFailSafeMode();

                
END_METHOD

METHOD describe
  VAR_INPUT
    executeContext : POINTER TO ExecuteContext;
  END_VAR
  VAR
    i : USINT;
  END_VAR
                  SUPER^.describe(executeContext);

IF (executeContext^.matchOption(cExecuteOptionSyntax)) THEN
	RETURN;
END_IF

IF (executeContext^.matchOption(cExecuteOptionParameter)) THEN	
	RETURN;
END_IF

executeContext^.appendPair('failsafe_active',gTypeHandler.getTokenForBool(PLC.FailSafeModeActive),FALSE,TRUE);
executeContext^.appendPair('systemstate',gTypeHandler.getTokenForEnum(cEnumTypeSystemState,SystemState.State),TRUE,TRUE);
executeContext^.appendPair('initialized',gTypeHandler.getTokenForBool(lInitialized),FALSE,TRUE);
executeContext^.appendPair('initialization_stage',SINT_TO_STRING(lInitializationStage),FALSE,TRUE);

IF (NOT(executeContext^.matchOption(cExecuteOptionChildren))) THEN
	RETURN;
END_IF

executeContext^.append(', ');
executeContext^.WriteStream^.increaseIndent();
executeContext^.formatWithNewlineIndent();
executeContext^.append('"subsystems": [');
executeContext^.WriteStream^.increaseIndent();

FOR i:=1 TO lSubsystemCount DO
	executeContext^.recordInitiatorWithNewlineIndent();
	executeContext^.appendPair('identity',lSubsystemSet[i]^.lIdentity,TRUE,FALSE);
	executeContext^.appendPair('type',lSubsystemSet[i]^.TypeToken,TRUE,TRUE);
	executeContext^.appendPair('subsystem',gTypeHandler.getTokenForEnum(cEnumTypeSubsystem,lSubsystemSet[i]^.SubSystem),TRUE,TRUE);
	executeContext^.recordTerminator();
	
	IF (i<lSubsystemCount) THEN
		executeContext^.append(', ');		
	END_IF
END_FOR

executeContext^.WriteStream^.decreaseIndent();
executeContext^.append(']');
executeContext^.WriteStream^.decreaseIndent();

                
END_METHOD

METHOD initializeStage0
                  //System REF= THIS^;

IF ((NOT(__ISVALIDREF(gSystemServices))) OR
	(NOT(__ISVALIDREF(_LocalMachine))) OR
	(NOT(__ISVALIDREF(_LEDDiagnostic))) OR
	(NOT(__ISVALIDREF(_ReportableChannelManager))) OR
	(NOT(__ISVALIDREF(_Executor))) OR
	(NOT(__ISVALIDREF(_Cycle))) OR
	(NOT(__ISVALIDREF(_PLC))) OR
	(NOT(__ISVALIDREF(_SystemState)))) THEN
	gCodeErrorHandler(pMessage:='null reference in system');
END_IF	

lVRTriggerClearFailSafeMode.initializeValueReference(lTriggerClearFailSafeMode,NopSelf,'ClearFailSafe','Trigger clearing failsafe mode','',cValueStyleTrigger);

initialize();

IF (gCodeErrorHandler.lState) THEN
	RETURN;
END_IF

lInitializationStage := 1;
                
END_METHOD

METHOD initializeSequence
                  IF (gCodeErrorHandler.lState) THEN
	RETURN;
END_IF

CASE (lInitializationStage) OF
	-1:
		preInitialize();

	0:
		initializeStage0();

	1:
		initializeStage1();
		
	2:
		initializeStage2();
	
	3:
		initializeStage3();
		
	4:
		postInitialize();
END_CASE
                
END_METHOD

METHOD initializeStage1
  VAR
    token : t_token_string;
  END_VAR
                  initialize();

token := 'true';
//eolus configure(sTokenFailSafeConfig,token,TRUE,0);

IF (gCodeErrorHandler.lState) THEN
	RETURN;
END_IF

lInitializationStage := 2;

                
END_METHOD

METHOD initializeStage2
  VAR
    token : t_token_string;
  END_VAR
                  initialize();

IF (gSystemServices.PLC.CrashSeverity<=4) THEN
	token := 'true';
	//eolus configure(sTokenFailSafeConfig,token,TRUE,0);
END_IF

IF (gCodeErrorHandler.lState) THEN
	RETURN;
END_IF

lInitializationStage := 3;

                
END_METHOD

METHOD initializeStage3
                  initialize();

IF (gCodeErrorHandler.lState) THEN
	RETURN;
END_IF

lInitializationStage := 4;


                
END_METHOD

METHOD configure
  VAR_INPUT
    executeContext : POINTER TO ExecuteContext;
  END_VAR
  VAR
    b : BOOL;
  END_VAR
                  IF (gSystemServices.Initialized) THEN
	IF (executeContext^.configureBool(cTokenFailSafeConfig,b,FALSE,0)) THEN
		RETURN;
	END_IF
END_IF

SUPER^.configure(executeContext);


                
END_METHOD

METHOD preInitialize
                  gTypeHandler.initialize();

gDebugFlags.Identifier := t_persistent_id.cPersistentID_DebugFlags;
gDebugFlags.initialize();

lInitializationStage := 0;
lFailSafeConfig := TRUE;

IF (gDebugFlags.Value := 16#FFFF) THEN
	gDebugFlags.Value := 0;
END_IF

                
END_METHOD

METHOD postInitialize
                  initialize();

IF ((PLC.CrashSeverity>0) AND (fCheckDebugFlags(cDebugEnableFailSafeOnCrash))) THEN
	gSystemServices.FailSafeMode := TRUE;
END_IF

PLC.setWatchdog();
PLC.executeAllCommands();

IF (gCodeErrorHandler.lState) THEN
	RETURN;
END_IF

lInitializationStage := 5;
lInitialized := TRUE;

                
END_METHOD

METHOD getParticle : POINTER TO t_particle
  VAR_INPUT
    name : REFERENCE TO t_token_string;
    id : t_particle_id;
  END_VAR
  VAR
    i : USINT;
    particle : t_particle_ptr;
  END_VAR
                  FOR i:=1 TO lSubsystemCount DO
	IF (id>0) THEN
		particle := lSubsystemSet[i]^.getParticle(name,id);
		IF (particle<>0) THEN
			getParticle := particle;
			RETURN;
		END_IF
	ELSE
		IF (strcmp(name,lSubsystemSet[i]^.lName)) THEN
			getParticle := lSubsystemSet[i];
			RETURN;
		END_IF		
	END_IF
END_FOR

getParticle := SUPER^.getParticle(name,id);

                
END_METHOD

METHOD registerSubsystem
  VAR_INPUT
    particle : t_particle_ptr;
  END_VAR
                  IF (particle=0) THEN
	RETURN;
END_IF

IF (lSubsystemCount>=cSubsystemSetMax) THEN
	gCodeErrorHandler(pMessage:='SubsystemSet overflow');
	RETURN;
END_IF

lSubsystemCount := lSubsystemCount + 1;
lSubsystemSet[lSubsystemCount] := particle;
particle^.Parent := 0;
particle^.lFeature := FALSE;

                
END_METHOD

PROPERTY LEDDiagnostic : REFERENCE TO LEDDiagnostic
GET
                    LEDDiagnostic ref= _LEDDiagnostic;
                  
END_GET
END_PROPERTY

PROPERTY TypeToken : t_medium_string
GET
                    TypeToken := 'System';
                  
END_GET
END_PROPERTY

PROPERTY Cycle : REFERENCE TO Cycle
GET
                    Cycle ref= _Cycle;
                  
END_GET
END_PROPERTY

PROPERTY ReportableChannelManager : REFERENCE TO ReportableChannelManager
GET
                    ReportableChannelManager ref= _ReportableChannelManager;
                  
END_GET
END_PROPERTY

PROPERTY SystemState : REFERENCE TO SystemState
GET
                    SystemState ref= _SystemState;
                  
END_GET
END_PROPERTY

PROPERTY LocalMachine : REFERENCE TO LocalMachine
GET
                    LocalMachine ref= _LocalMachine;
                  
END_GET
END_PROPERTY

PROPERTY PLC : REFERENCE TO PLC
GET
                    PLC ref= _PLC;
                  
END_GET
END_PROPERTY

PROPERTY Initialized : BOOL
GET
                    Initialized := lInitialized;
                  
END_GET
END_PROPERTY

PROPERTY Executor : REFERENCE TO Executor
GET
                    Executor ref= _Executor;
                  
END_GET
END_PROPERTY
END_FUNCTION_BLOCK

FUNCTION_BLOCK SystemState EXTENDS NonOperationalParticleSet
  VAR CONSTANT
    cEventTimerPeriod : t_time := TIME#1m0s0ms;
    cPoweringUpPeriod : t_time := TIME#2s0ms;
    cExitOperationalPeriod : t_time := TIME#6s0ms;
  END_VAR
  VAR
    lState : ValueObjectEnumType;
    lPreviousState : t_system_state := cSystemStateNone;
    lChargingEnabled : BOOL := FALSE;
    lTransitionEstopState : t_system_state := cSystemStatePreparing;
    lPoweringUpTimer : t_timer;
    lExitOperationalTimer : t_timer;
    lTransitionFlag : BOOL := FALSE;
    lInitializedCounter : USINT := 0;
    lStateCounterInitialized : USINT := 0;
    lStateCounterStandby : USINT := 0;
    lStateCounterCharging : USINT := 0;
    lStateCounterPreparing : USINT := 0;
    lStateCounterPreOperational : USINT := 0;
    lStateCounterPoweringDown : USINT := 0;
    lStateCounterPoweringUp : USINT := 0;
    lStateCounterExitOperational : USINT := 0;
    lStateCounterGoOperational : USINT := 0;
    lStateCounterOperational : USINT := 0;
    lSystemControlTrace : ReportableContextSystemControl;
    lAllowUpTrace : ReportableContextSystemStateUp;
    lAllowDownTrace : ReportableContextSystemStateDown;
    lForceMaxTrace : ReportableContextSystemStateUp;
    lNextStateTrace : ReportableContextSystemStateUp;
    lTransitionInitializedStandby : ReportableEvent;
    lTransitionStandbyPreparing : ReportableEvent;
    lTransitionStandbyInitialized : ReportableEvent;
    lTransitionPreparingPreOperational : ReportableEvent;
    lTransitionPreparingCharging : ReportableEvent;
    lTransitionPreparingStandby : ReportableEvent;
    lTransitionChargingPreparing : ReportableEvent;
    lTransitionPreOperationalPreparing : ReportableEvent;
    lTransitionPoweringUpGoOperational : ReportableEvent;
    lTransitionGoOperationalOperational : ReportableEvent;
    lTransitionExitOperationalPoweringDown : ReportableEvent;
    lTransitionPoweringDownPreOperational : ReportableEvent;
    lAutomaticStart : BOOL := FALSE;
    lCausalAutomaticStart : ReportableCausal;
  END_VAR

            ;
          

METHOD initialize
                  lState.EnumType := cEnumTypeSystemState;
lState.initializeValueObject(NopSelf,'State','System state','',cValueStyleConfigurable);

lSystemControlTrace.initializeEvent(NopSelf,'',cECSystemControl);
lAllowUpTrace.initializeEvent(NopSelf,'',cECAllowUpState);
lAllowDownTrace.initializeEvent(NopSelf,'',cECAllowDownState);
lForceMaxTrace.initializeEvent(NopSelf,'',cECForceMaxState);
lNextStateTrace.initializeEvent(NopSelf,'',cECNextState);

lTransitionInitializedStandby.initializeEvent(NopSelf,'',cECTransitionInitializedStandby);
lTransitionStandbyPreparing.initializeEvent(NopSelf,'',cECTransitionStandbyPreparing);
lTransitionStandbyInitialized.initializeEvent(NopSelf,'',cECTransitionStandbyInitialized);
lTransitionPreparingPreOperational.initializeEvent(NopSelf,'',cECTransitionPreparingPreOperational);
lTransitionPreparingCharging.initializeEvent(NopSelf,'',cECTransitionPreparingCharging);
lTransitionPreparingStandby.initializeEvent(NopSelf,'',cECTransitionPreparingStandby);
lTransitionChargingPreparing.initializeEvent(NopSelf,'',cECTransitionChargingPreparing);
lTransitionPreOperationalPreparing.initializeEvent(NopSelf,'',cECTransitionPreOperationalPreparing);
lTransitionPoweringUpGoOperational.initializeEvent(NopSelf,'',cECTransitionPoweringUpGoOperational);
lTransitionGoOperationalOperational.initializeEvent(NopSelf,'',cECTransitionGoOperationalOperational);
lTransitionExitOperationalPoweringDown.initializeEvent(NopSelf,'',cECTransitionExitOperationalPoweringDown);
lTransitionPoweringDownPreOperational.initializeEvent(NopSelf,'',cECTransitionPoweringDownPreOperational);

lCausalAutomaticStart.initializeState(NopSelf,'',cCCAutomaticStart);

SUPER^.initialize();

// lTransitionEstopState := cSystemStateInitialized;
lTransitionEstopState := cSystemStatePreparing;

lPoweringUpTimer.initialize();
lPoweringUpTimer.Enable := TRUE;
lPoweringUpTimer.Period := cPoweringUpPeriod;

lExitOperationalTimer.initialize();
lExitOperationalTimer.Enable := TRUE;
lExitOperationalTimer.Period := cExitOperationalPeriod;

lState.Value := cSystemStateInitialized;
lPreviousState := State;

lTransitionFlag := FALSE;
lChargingEnabled := FALSE;

lTransitionInitializedStandby.Suppress := FALSE;
lTransitionStandbyPreparing.Suppress := false;
lTransitionStandbyInitialized.Suppress := false;
lTransitionPreparingPreOperational.Suppress := false;
lTransitionPreparingCharging.Suppress := false;
lTransitionPreparingStandby.Suppress := false;
lTransitionChargingPreparing.Suppress := false;
lTransitionPreOperationalPreparing.Suppress := false;
lTransitionPoweringUpGoOperational.Suppress := false;
lTransitionGoOperationalOperational.Suppress := false;
lTransitionExitOperationalPoweringDown.Suppress := false;
lTransitionPoweringDownPreOperational.Suppress := false;


                
END_METHOD

METHOD operator
                  lSystemControlTrace.operator();
lSystemControlTrace.apply();

lAllowUpTrace.operator();
lAllowDownTrace.operator();

IF (State<=cSystemStateStandby) THEN
	gSystemServices.LEDDiagnostic.Code := cLEDCodeStandby;
ELSE
	gSystemServices.LEDDiagnostic.Code := cLEDCodeNormal;	
END_IF

CASE State OF
	cSystemStateNone:
		;
	cSystemStateInitialized:
		stateInitialized();
	cSystemStateStandby:
		stateStandby();
	cSystemStatePreparing:
		statePreparing();
	cSystemStateCharging:
		stateCharging();
	cSystemStatePreOperational:
		statePreOperational();
	cSystemStatePoweringDown:
		statePoweringDown();
	cSystemStatePoweringUp:
		statePoweringUp();
	cSystemStateGoOperational:
		stateGoOperational();
	cSystemStateExitOperational:
		stateExitOperational();
	cSystemStateOperational:
		stateOperational();
END_CASE

lForceMaxTrace.operator();

IF (lNextStateTrace.check(State)>lForceMaxTrace.State) THEN
	transitionNextState(lForceMaxTrace.State,ADR(lForceMaxTrace),lForceMaxTrace.Override);
END_IF

lNextStateTrace.operator();
lPreviousState := lState.Value;
lState.Value := lNextStateTrace.update(State);
lState.operator();

                
END_METHOD

METHOD request
  VAR_INPUT
    requestedSystemMethod : t_system_method;
  END_VAR
                  
                
END_METHOD

METHOD stateCharging
                  lStateCounterCharging := lStateCounterCharging + 1;

(* up - no automatic transitions *)
;

(* down *)
IF (lForceMaxTrace.State<cSystemStateCharging) THEN
	lTransitionChargingPreparing.trigger(FALSE);
	transitionNextState(cSystemStatePreparing,ADR(lTransitionChargingPreparing),FALSE);
END_IF

                
END_METHOD

METHOD stateExitOperational
                  lStateCounterExitOperational := lStateCounterExitOperational + 1;

lExitOperationalTimer.operator();

(* up - no automatic transitions *)

(* down *)
IF ((lAllowDownTrace.State<=cSystemStatePoweringDown) AND
	(lExitOperationalTimer.Expired)) THEN
	lTransitionExitOperationalPoweringDown.trigger(FALSE);
	transitionNextState(cSystemStatePoweringDown,ADR(lTransitionExitOperationalPoweringDown),FALSE);
END_IF

                
END_METHOD

METHOD stateGoOperational
                  lStateCounterGoOperational := lStateCounterGoOperational + 1;

(* up *)
IF (lAllowUpTrace.State>=cSystemStateOperational) THEN
	lTransitionGoOperationalOperational.trigger(FALSE);
	transitionNextState(cSystemStateOperational,ADR(lTransitionGoOperationalOperational),FALSE);
END_IF

(* down - no automatic down *)
                
END_METHOD

METHOD stateInitialized
                  lStateCounterInitialized := lStateCounterInitialized + 1;

(* up *)
IF (lAllowUpTrace.State>=cSystemStateStandby) THEN
	lTransitionInitializedStandby.trigger(FALSE);
	transitionNextState(cSystemStateStandby,ADR(lTransitionInitializedStandby),FALSE);
END_IF

(* no down *)

IF (lTransitionFlag) THEN
	lInitializedCounter := lInitializedCounter + 1;
END_IF
                
END_METHOD

METHOD stateOperational
                  lStateCounterOperational := lStateCounterOperational + 1;

lExitOperationalTimer.reset();

(* up - no automatic transitions *)
;

(* down - no automatic transitions *)
;
                
END_METHOD

METHOD statePoweringDown
                  lStateCounterPoweringDown := lStateCounterPoweringDown + 1;

(* up - no automatic transitions *)

(* down *)
IF (lAllowDownTrace.State<=cSystemStatePreOperational) THEN
	lTransitionPoweringDownPreOperational.trigger(FALSE);
	transitionNextState(cSystemStatePreOperational,ADR(lTransitionPoweringDownPreOperational),FALSE);
END_IF
                
END_METHOD

METHOD statePoweringUp
                  lStateCounterPoweringUp := lStateCounterPoweringUp + 1;

lPoweringUpTimer.operator();

(* up *)
IF ((lAllowUpTrace.State>=cSystemStateGoOperational) AND
	(lPoweringUpTimer.Expired)) THEN
	lTransitionPoweringUpGoOperational.trigger(FALSE);
	transitionNextState(cSystemStateGoOperational,ADR(lTransitionPoweringUpGoOperational),FALSE);
END_IF

(* down - no automatic down *)
                
END_METHOD

METHOD statePreOperational
                  lStateCounterPreOperational := lStateCounterPreOperational + 1;

lPoweringUpTimer.reset();

(* up *)
IF (lAutomaticStart) THEN
	lCausalAutomaticStart.trigger(FALSE);
	transitionStart(cSystemStateOperational,ADR(lCausalAutomaticStart),lCausalAutomaticStart.Override);
END_IF

(* down *)
IF (lForceMaxTrace.State<cSystemStatePreOperational) THEN
	lTransitionPreOperationalPreparing.trigger(FALSE);
	transitionNextState(cSystemStatePreparing,ADR(lTransitionPreOperationalPreparing),FALSE);
END_IF
                
END_METHOD

METHOD statePreparing
                  lStateCounterPreparing := lStateCounterPreparing + 1;

(* up *)
IF (lAllowUpTrace.State>=cSystemStatePreOperational) THEN
	lTransitionPreparingPreOperational.trigger(FALSE);
	transitionNextState(cSystemStatePreOperational,ADR(lTransitionPreparingPreOperational),FALSE);
END_IF

IF ((lAllowUpTrace.State=cSystemStateCharging) AND
	(lChargingEnabled)) THEN
	lTransitionPreparingCharging.trigger(FALSE);
	transitionNextState(cSystemStateCharging,ADR(lTransitionPreparingCharging),FALSE);
END_IF

(* down *)
IF (lForceMaxTrace.State<cSystemStatePreparing) THEN
	lTransitionPreparingStandby.trigger(FALSE);
	transitionNextState(cSystemStateStandby,ADR(lTransitionPreparingStandby),FALSE);
END_IF
                
END_METHOD

METHOD stateStandby
                  lStateCounterStandby := lStateCounterStandby + 1;

(* up *)
IF (lAllowUpTrace.State>=cSystemStatePreparing) THEN
	lTransitionStandbyPreparing.trigger(FALSE);
	transitionNextState(cSystemStatePreparing,ADR(lTransitionStandbyPreparing),FALSE);
END_IF

(* down *)
IF (lForceMaxTrace.State<cSystemStateStandby) THEN
	lTransitionStandbyInitialized.trigger(FALSE);
	transitionNextState(cSystemStateInitialized,ADR(lTransitionStandbyInitialized),FALSE);
END_IF
                
END_METHOD

METHOD transitionAllowDown
  VAR_INPUT
    allowable : t_system_state;
    reportable : POINTER TO t_reportable;
    override : BOOL;
  END_VAR
                  lAllowDownTrace.process(allowable,reportable,override);
                
END_METHOD

METHOD transitionAllowUp
  VAR_INPUT
    allowable : t_system_state;
    reportable : POINTER TO t_reportable;
    override : BOOL;
  END_VAR
                  lAllowUpTrace.process(allowable,reportable,override);

                
END_METHOD

METHOD transitionEstop
  VAR_INPUT
    allowable : t_system_state;
    reportable : POINTER TO t_reportable;
    override : BOOL;
  END_VAR
                  IF (State>cSystemStatePreOperational) THEN	
	transitionNextState(lTransitionEstopState,reportable,override);
END_IF

transitionAllowUp(allowable,reportable,override);
transitionForceMax(allowable,reportable,override);

                
END_METHOD

METHOD transitionForceMax
  VAR_INPUT
    allowable : t_system_state;
    reportable : POINTER TO t_reportable;
    override : BOOL;
  END_VAR
                  lForceMaxTrace.process(allowable,reportable,override);
                
END_METHOD

METHOD transitionInitialized
  VAR_INPUT
    allowable : t_system_state;
    reportable : POINTER TO t_reportable;
    override : BOOL;
  END_VAR
                  IF (State<=cSystemStatePreOperational) THEN	
	transitionNextState(cSystemStateInitialized,reportable,override);
END_IF

transitionAllowUp(allowable,reportable,override);
transitionForceMax(allowable,reportable,override);

                
END_METHOD

METHOD transitionNextState
  VAR_INPUT
    nextState : t_system_state;
    reportable : POINTER TO t_reportable;
    override : BOOL;
  END_VAR
                  lNextStateTrace.process(nextState,reportable,override);

                
END_METHOD

METHOD transitionStart
  VAR_INPUT
    allowable : t_system_state;
    reportable : POINTER TO t_reportable;
    override : BOOL;
  END_VAR
                  IF (State=cSystemStatePreOperational) THEN
	transitionNextState(cSystemStatePoweringUp,reportable,override);
	transitionAllowUp(allowable,reportable,override);
END_IF

                
END_METHOD

METHOD transitionStop
  VAR_INPUT
    allowable : t_system_state;
    reportable : POINTER TO t_reportable;
    override : BOOL;
  END_VAR
                  IF (State>cSystemStatePreOperational) THEN
	IF (State>cSystemStatePoweringUp) THEN		
		transitionNextState(cSystemStateExitOperational,reportable,override);
		transitionForceMax(cSystemStateExitOperational,reportable,override);

	ELSIF (State>cSystemStatePreOperational) THEN		
		transitionNextState(cSystemStatePoweringDown,reportable,override);
		transitionForceMax(cSystemStatePoweringDown,reportable,override);
	END_IF
	
	RETURN;
END_IF

transitionAllowUp(allowable,reportable,override);
transitionForceMax(allowable,reportable,override);

                
END_METHOD

PROPERTY ChargingEnabled : BOOL
GET
                    ChargingEnabled := lChargingEnabled;
                  
END_GET
SET
                    lChargingEnabled := ChargingEnabled;
                  
END_SET
END_PROPERTY

(* {attribute 'monitoring' := 'call'} *)
PROPERTY State : t_system_state
GET
                    State := lState.Value;
                  
END_GET
END_PROPERTY

PROPERTY SystemControl : REFERENCE TO ReportableContextSystemControl
GET
                    SystemControl ref= lSystemControlTrace;
                  
END_GET
END_PROPERTY

PROPERTY TypeToken : t_medium_string
GET
                    TypeToken := 'SystemState';
                  
END_GET
END_PROPERTY

PROPERTY AutomaticStart : BOOL
GET
                    AutomaticStart := lAutomaticStart;
                  
END_GET
SET
                    lAutomaticStart := AutomaticStart;
                  
END_SET
END_PROPERTY
END_FUNCTION_BLOCK

FUNCTION_BLOCK ConnectionHandler
  VAR
    lEnabled : BOOL := TRUE;
    lInteractive : BOOL := TRUE;
    lConnection : POINTER TO TCPConnection := 0;
    lCount : UINT := 0;
  END_VAR

            
          

METHOD operator
                  

                
END_METHOD

METHOD prompt
                  
                
END_METHOD

METHOD connecting
  VAR
    str : t_long_string;
  END_VAR
                  IF (NOT(lInteractive)) THEN
	RETURN;
END_IF

str := CONCAT('Connected to <',
	CONCAT(gSystemServices.LocalMachine.MachineName,
	CONCAT('> at time <',
	CONCAT(gSystemServices.Cycle.SystemTime,'>$r$n'))));

lConnection^.write(ADR(str[0]),INT_TO_UINT(LEN(str)) + 1);

prompt();




                
END_METHOD

PROPERTY Connection : POINTER TO TCPConnection
GET
                    Connection := lConnection;
                  
END_GET
SET
                    lConnection := Connection;
                  
END_SET
END_PROPERTY

PROPERTY Enabled : BOOL
GET
                    Enabled := lEnabled;

                  
END_GET
SET
                    lEnabled := Enabled;
                  
END_SET
END_PROPERTY

PROPERTY Interactive : BOOL
GET
                    Interactive := lInteractive;
                  
END_GET
SET
                    lInteractive := Interactive;


                  
END_SET
END_PROPERTY
END_FUNCTION_BLOCK

FUNCTION_BLOCK EchoConnectionHandler EXTENDS ConnectionHandler
  VAR
    lReadStream : t_stream;
  END_VAR

            
          

METHOD operator
                  IF (NOT(lConnection^.read(ADR(lReadStream)))) THEN
	RETURN;
END_IF

lCount := lCount + 1;

IF (NOT(lEnabled)) THEN
	RETURN;
END_IF

lReadStream.terminateWithNewline();
lConnection^.write(lReadStream.Buffer,lReadStream.Length);
prompt();

                
END_METHOD

METHOD prompt
  VAR
    str : t_medium_string;
  END_VAR
                  str := CONCAT(gSystemServices.LocalMachine.MachineName,' echo>');
lConnection^.write(ADR(str[0]),INT_TO_UINT(LEN(str)) + 1);

                
END_METHOD

METHOD connecting
                  SUPER^.connecting();

prompt();

	
                
END_METHOD
END_FUNCTION_BLOCK

FUNCTION_BLOCK ParseConnectionHandler EXTENDS ConnectionHandler
  VAR CONSTANT
    cParseMaxTokens : USINT := 32;
  END_VAR
  VAR
    lReadStream : t_stream;
    lExecuteContext : ExecuteContextParse;
    lCurrentCommand : t_command_request;
    lParsingComplete : BOOL := TRUE;
    lPromptRequired : BOOL := TRUE;
    lTokensParsedCount : USINT := 0;
  END_VAR

            
          

METHOD prompt
                  IF (NOT(lInteractive)) THEN
	RETURN;
END_IF

//str := CONCAT(gSystemServices.LocalMachine.MachineName,' $$>');
lExecuteContext.append('$$>');

                
END_METHOD

METHOD connecting
                  SUPER^.connecting();

clear();

                
END_METHOD

METHOD operator
  VAR
    i : USINT;
  END_VAR
                  lExecuteContext.operator();
lConnection^.write(lExecuteContext.WriteStream^.Buffer,lExecuteContext.WriteStream^.Length);

IF ((lParsingComplete) OR
	(NOT(lEnabled))) THEN
	IF (NOT(lConnection^.read(ADR(lReadStream)))) THEN
		RETURN;
	END_IF

	lCount := lCount + 1;
	
	IF (NOT(lEnabled)) THEN
		clear();
		RETURN;
	END_IF

	lParsingComplete := FALSE;
	lReadStream.initializeParsing();
END_IF

                
END_METHOD

METHOD initialize
                  lExecuteContext.Source REF= THIS^;

lExecuteContext.WriteStream^.IndentStr := '';
lExecuteContext.WriteStream^.NewlineStr := '$n';
lExecuteContext.WriteStream^.RecordInitiatorStr := '{';
lExecuteContext.WriteStream^.RecordTerminatorStr := '}';

                
END_METHOD

METHOD clear
                  lReadStream.clear();

lParsingComplete := TRUE;

                
END_METHOD

METHOD getNextExecuteCommand : BOOL
  VAR_INPUT
    command : REFERENCE TO t_command_request;
  END_VAR
                  IF (lPromptRequired) THEN
	prompt();
	lPromptRequired := FALSE;
END_IF

getNextExecuteCommand := parse(command);

IF (NOT(getNextExecuteCommand)) THEN
	RETURN;
END_IF

lPromptRequired := TRUE;

if (lExecuteContext.Error) then
	RETURN;
END_IF

IF ((command.particle=0) OR
	(command.command=cTokenNone)) THEN
	lExecuteContext.ExecuteReturn := cExecuteReturnExecutionSyntaxIncompleteRequest;
	lExecuteContext.Error := TRUE;
END_IF

                
END_METHOD

METHOD parse : BOOL
  VAR_INPUT
    command : REFERENCE TO t_command_request;
  END_VAR
  VAR
    parseTokenType : t_parse_token_type;
    token : t_fqtoken_string;
    parameter : t_token_type;
    value : t_token_string;
    option : t_execute_option;
    name : POINTER TO t_particle;
    i : USINT;
    parameterPending : BOOL := FALSE;
    namePending : BOOL := FALSE;
  END_VAR
                  parse := FALSE;

command.particle := 0;
command.command := cTokenNone;
command.argumentCount := 0;
command.optionCount := 0;

IF (lParsingComplete) THEN
	RETURN;
END_IF

name := ADR(gSystemServices);

FOR lTokensParsedCount:=0 TO cParseMaxTokens DO
	parseTokenType := lReadStream.getNextToken(ADR(token));
	
	IF ((parseTokenType=cParseTokenNone) OR
		(parseTokenType=cParseTokenFinished)) THEN
		lParsingComplete := TRUE;
		RETURN;		
	END_IF

	IF (parseTokenType=cParseTokenTerminator) THEN
		RETURN;		
	END_IF
	
	parse := TRUE;
	
	IF (parseTokenType=cParseTokenOverflow) THEN
		lExecuteContext.ExecuteReturn := cExecuteReturnExecutionSyntaxTokenOverflow;
		lExecuteContext.Error := TRUE;
		lReadStream.skipOverError();
		RETURN;		
	END_IF

	IF (parseTokenType=cParseTokenError) THEN
		lExecuteContext.ExecuteReturn := cExecuteReturnExecutionSyntax;
		lExecuteContext.Error := TRUE;
		lReadStream.skipOverError();
		RETURN;		
	END_IF
	
	IF ((parameterPending) AND
		(parseTokenType<>cParseTokenName) AND
		(parseTokenType<>cParseTokenSimple)) THEN
		lExecuteContext.ExecuteReturn := cExecuteReturnExecutionSyntaxIncompleteParameter;
		lExecuteContext.Error := TRUE;
		lReadStream.skipOverError();
		RETURN;						
	END_IF
	
	IF ((namePending) AND
		(parseTokenType<>cParseTokenName) AND
		(parseTokenType<>cParseTokenSimple)) THEN
		lExecuteContext.ExecuteReturn := cExecuteReturnExecutionSyntaxIncompleteName;
		lExecuteContext.Error := TRUE;
		lReadStream.skipOverError();
		RETURN;						
	END_IF

	IF ((command.particle=0) AND
		(parseTokenType<>cParseTokenName) AND
		(parseTokenType<>cParseTokenSimple)) THEN
		lExecuteContext.ExecuteReturn := cExecuteReturnExecutionSyntaxStartWithName;
		lExecuteContext.Error := TRUE;
		lReadStream.skipOverError();
		RETURN;						
	END_IF
	
	IF ((command.command=cTokenNone) AND
		(parseTokenType<>cParseTokenName) AND
		(parseTokenType<>cParseTokenSimple)) THEN
		lExecuteContext.ExecuteReturn := cExecuteReturnExecutionSyntaxCommandAfterName;
		lExecuteContext.Error := TRUE;
		lReadStream.skipOverError();
		RETURN;						
	END_IF
	
	CASE parseTokenType OF
		cParseTokenName:
			name := getParticle(name,token);
			IF (name=0) THEN
				lExecuteContext.ExecuteReturn := cExecuteReturnExecutionSyntaxUnkownName;
				lExecuteContext.Error := TRUE;
				lReadStream.skipOverError();
				RETURN;	
			END_IF

			namePending := TRUE;						
									
		cParseTokenSimple:
			IF (command.particle=0) THEN
				command.particle := getParticle(name,token);

				IF (command.particle=0) THEN
					lExecuteContext.ExecuteReturn := cExecuteReturnExecutionSyntaxUnkownName;
					lExecuteContext.Error := TRUE;
					lReadStream.skipOverError();
					RETURN;	
				END_IF								
					
				namePending := FALSE;
				name := ADR(gSystemServices);

				CONTINUE;
			END_IF

			IF (parameterPending) THEN
				IF (namePending) THEN
					name := getParticle(name,token);

					IF (name=0) THEN
						lExecuteContext.ExecuteReturn := cExecuteReturnExecutionSyntaxUnkownNameForParameter;
						lExecuteContext.Error := TRUE;
						lReadStream.skipOverError();
						RETURN;	
					END_IF
					
					value := gTypeHandler.getTokenForUINT(name^.lParticleId);

					namePending := FALSE;
					name := ADR(gSystemServices);
				ELSE
					value := token;
				END_IF								
	
				IF (command.argumentCount>=cExecuteArgumentListCount) THEN
					lExecuteContext.ExecuteReturn := cExecuteReturnTooManyArguments;
					lExecuteContext.Error := TRUE;
					lReadStream.skipOverError();
					RETURN;				
				END_IF
			
				command.argumentCount := command.argumentCount + 1;
				command.arguments[command.argumentCount].parameter := parameter;
				command.arguments[command.argumentCount].value := value;
				command.arguments[command.argumentCount].processed := FALSE;
				
				CONTINUE;
			END_IF			

			IF (command.command<>cTokenNone) THEN
				lExecuteContext.ExecuteReturn := cExecuteReturnExecutionSyntaxDuplicateCommands;
				lExecuteContext.Error := TRUE;
				lReadStream.skipOverError();
				RETURN;				
			END_IF

			IF (NOT(gTypeHandler.getEnumFromToken(cEnumTypeTokenType,token,command.command))) THEN
				lExecuteContext.ExecuteReturn := cExecuteReturnUnknownCommand;
				lExecuteContext.Error := TRUE;
				lReadStream.skipOverError();
				RETURN;
			END_IF			
			
		cParseTokenParameter:	
			IF (NOT(gTypeHandler.getEnumFromToken(cEnumTypeTokenType,token,parameter))) THEN
				lExecuteContext.ExecuteReturn := cExecuteReturnUnknownParameter;
				lExecuteContext.Error := TRUE;
				lReadStream.skipOverError();
				RETURN;						
			END_IF

			parameterPending := TRUE;

		cParseTokenOption:
			IF (NOT(gTypeHandler.getEnumFromToken(cEnumTypeExecuteOption,token,option))) THEN
				lExecuteContext.ExecuteReturn := cExecuteReturnUnknownOption;
				lExecuteContext.Error := TRUE;
				lReadStream.skipOverError();
				RETURN;
			END_IF
			
			IF (command.optionCount>=cExecuteOptionListCount) THEN
				lExecuteContext.ExecuteReturn := cExecuteReturnExecutionSyntaxTooManyOptions;
				lExecuteContext.Error := TRUE;
				lReadStream.skipOverError();
				RETURN;				
			END_IF
			
			command.optionCount := command.optionCount + 1;
			command.options[command.optionCount] := option;
	END_CASE
END_FOR

lExecuteContext.ExecuteReturn := cExecuteReturnExecutionSyntaxUnbounded;
lExecuteContext.Error := TRUE;
lReadStream.skipOverError();

                
END_METHOD

METHOD getParticle : POINTER TO t_particle
  VAR_INPUT
    particle : POINTER TO t_particle;
    fqn : t_fqtoken_string;
  END_VAR
  VAR
    tokens : t_token_string_set;
    count : USINT := 0;
    i : USINT;
  END_VAR
                  IF (particle=0) THEN
	getParticle := 0;
	RETURN;
END_IF

IF (NOT(splitFQN(fqn,tokens,count))) THEN
	getParticle := 0;
	RETURN;
END_IF

IF (count=0) THEN
	getParticle := 0;
	RETURN;
END_IF

IF (count=1) THEN
	getParticle := particle^.getParticle(tokens[1],0);
	RETURN;
END_IF

IF (particle<>ADR(gSystemServices)) THEN
	getParticle := 0;
	RETURN;	
END_IF

IF (NOT(tokens[1]=gNameSpace)) THEN
	getParticle := 0;
	RETURN;
END_IF

FOR i:=2 TO count DO
	particle := particle^.getParticle(tokens[i],0);
	
	IF (particle=0) THEN
		getParticle := 0;
		RETURN;		
	END_IF	
END_FOR

getParticle := particle;

                
END_METHOD

PROPERTY ReadWrite : BOOL
GET
                    ReadWrite := lExecuteContext.ReadWrite;
                  
END_GET
SET
  VAR
    i : USINT;
  END_VAR
                    lExecuteContext.ReadWrite := ReadWrite;

                  
END_SET
END_PROPERTY

PROPERTY ExecuteContext : POINTER TO ExecuteContextParse
GET
                    ExecuteContext:= ADR(lExecuteContext);
                  
END_GET
END_PROPERTY
END_FUNCTION_BLOCK

FUNCTION_BLOCK ReportableChannelClientTCP EXTENDS ReportableChannel
  VAR CONSTANT
    cCycleCount : USINT := 2;
    cCyclePeriod : t_time := TIME#3m0s0ms;
  END_VAR
  VAR
    lClient : TCPClient;
    lExecuteContext : ExecuteContext;
    lVolumeMbs : REAL;
    lVolumeBits : UDINT;
    lCycleTimer : t_timer;
    lCycleIndex : UINT := 0;
    lCycleCount : USINT := cCycleCount;
  END_VAR

            
          

METHOD initialize
                  registerOperational(ADR(lClient));

SUPER^.initialize();

lExecuteContext.WriteStream^.IndentStr := '';
lExecuteContext.WriteStream^.NewlineStr := '$n';
lExecuteContext.WriteStream^.RecordInitiatorStr := '{';
lExecuteContext.WriteStream^.RecordTerminatorStr := '}';

lExecuteContext.WriteStream^.clear();

lCycleIndex := 0;

lCycleTimer.initialize();
lCycleTimer.Enable := TRUE;
lCycleTimer.Period := cCyclePeriod;


                
END_METHOD

METHOD _reportEvent
  VAR_INPUT
    event : POINTER TO t_reportableevent;
  END_VAR
                  lExecuteContext.recordInitiator();
event^.describe(ADR(lExecuteContext));
lExecuteContext.recordTerminatorWithNewline();

                
END_METHOD

METHOD _reportState
  VAR_INPUT
    state : POINTER TO t_reportablestate;
    expired : BOOL;
  END_VAR
  VAR
    lengthA : UINT;
    lengthB : UINT;
  END_VAR
                  lExecuteContext.recordInitiator();
state^.describe(ADR(lExecuteContext));
lExecuteContext.recordTerminatorWithNewline();


                
END_METHOD

METHOD _reportStateExpired
  VAR_INPUT
    state : POINTER TO t_reportablestate;
  END_VAR
                  _reportState(state);

                
END_METHOD

METHOD operator
  VAR
    i : USINT;
    state : POINTER TO t_reportablestate;
    length : UINT;
  END_VAR
                  lCycleTimer.operator();
IF (lCycleTimer.Expired) THEN
	lCycleTimer.reset();
	lCycleIndex := 1;
END_IF

i := 0;
WHILE ((lCycleIndex>0) AND (i<lCycleCount)) DO
	i := i + 1;
	
	state := lReportableChannelManager^.lReportableStateManager.cycle(lChannelMask,ADR(lCycleIndex),FALSE);
	IF (state<>0) THEN
		_reportState(state,FALSE);	
	END_IF
END_WHILE

IF (gSystemServices.Cycle.IntegralClockTick) THEN
	lVolumeMbs := UDINT_TO_REAL(lVolumeBits)/1000000.0;
	lVolumeBits := 0;
END_IF

SUPER^.operator();

length := lExecuteContext.WriteStream^.Length;
	
IF (lEnabled) THEN
	lClient.write(lExecuteContext.WriteStream^.Buffer,length);
	lVolumeBits := lVolumeBits + length;
END_IF

lExecuteContext.WriteStream^.clear();

                
END_METHOD

METHOD header
                  (*lStream.newline();
lStream.append('timestep <');
lStream.append(System.Cycle.SystemTime);
lStream.append('> state <');
lStream.append(gTypeHandler.getTokenForEnum(cEnumTypeSystemState,gSystemServices.SystemState.State));
lStream.append('>');*)

lStream.append('{"timestep":"');
lStream.append(System.Cycle.SystemTime);
lStream.append('","state":"');
lStream.append(gTypeHandler.getTokenForEnum(cEnumTypeSystemState,gSystemServices.SystemState.State));
lStream.append('",');

                
END_METHOD

METHOD _reportStateActiveRising
  VAR_INPUT
    state : POINTER TO t_reportablestate;
  END_VAR
                  _reportState(state);




                
END_METHOD

PROPERTY VolumeMbs : REAL
GET
                    VolumeMbs := lVolumeMbs;
                  
END_GET
END_PROPERTY

PROPERTY TypeToken : t_medium_string
GET
                    TypeToken := 'RepChanClientTCP';
                  
END_GET
END_PROPERTY

PROPERTY Client : REFERENCE TO TCPClient
GET
                    Client ref= lClient;
                  
END_GET
END_PROPERTY

PROPERTY ChannelConnected : BOOL
GET
                    ChannelConnected := lClient.ClientConnected;

                  
END_GET
END_PROPERTY
END_FUNCTION_BLOCK

FUNCTION_BLOCK ReportableChannelLogTCP EXTENDS ReportableChannel
  VAR
    lServer : NullTCPServer;
    lExecuteContext : ExecuteContext;
    lVolumeMbs : REAL;
    lVolumeBits : UDINT;
  END_VAR

            
          

METHOD initialize
                  registerOperational(ADR(lServer));

SUPER^.initialize();

lExecuteContext.WriteStream^.IndentStr := '';
lExecuteContext.WriteStream^.NewlineStr := '$n';
lExecuteContext.WriteStream^.RecordInitiatorStr := '{';
lExecuteContext.WriteStream^.RecordTerminatorStr := '}';

lExecuteContext.WriteStream^.clear();

                
END_METHOD

METHOD _reportEvent
  VAR_INPUT
    event : POINTER TO t_reportableevent;
  END_VAR
  VAR
    i : USINT;
  END_VAR
                  IF (lExecuteContext.WriteStream^.Length=0) THEN
	header();
END_IF

lExecuteContext.recordInitiator();
event^.describe(ADR(lExecuteContext));
lExecuteContext.recordTerminatorWithNewline();

                
END_METHOD

METHOD _reportState
  VAR_INPUT
    state : POINTER TO t_reportablestate;
    expired : BOOL;
  END_VAR
  VAR
    i : USINT;
  END_VAR
                  IF (lExecuteContext.WriteStream^.Length=0) THEN
	header();
END_IF

lExecuteContext.recordInitiator();
state^.describe(ADR(lExecuteContext));
lExecuteContext.recordTerminatorWithNewline();

                
END_METHOD

METHOD _reportStateExpired
  VAR_INPUT
    state : POINTER TO t_reportablestate;
  END_VAR
  VAR
    i : USINT;
  END_VAR
                  _reportState(state);


                
END_METHOD

METHOD operator
  VAR
    length : UINT;
  END_VAR
                  IF (gSystemServices.Cycle.IntegralClockTick) THEN
	lVolumeMbs := UDINT_TO_REAL(lVolumeBits)/1000000.0;
	lVolumeBits := 0;
END_IF

SUPER^.operator();

length := lExecuteContext.WriteStream^.Length;
	
IF (lEnabled) THEN
	lServer.write(lExecuteContext.WriteStream^.Buffer,length);
	lVolumeBits := lVolumeBits + length;
END_IF

lExecuteContext.WriteStream^.clear();

                
END_METHOD

METHOD header
                  lExecuteContext.WriteStream^.newline();
lExecuteContext.WriteStream^.append('timestep <');
lExecuteContext.WriteStream^.append(gSystemServices.Cycle.SystemTime);
lExecuteContext.WriteStream^.append('> state <');
lExecuteContext.WriteStream^.append(gTypeHandler.getTokenForEnum(cEnumTypeSystemState,gSystemServices.SystemState.State));
lExecuteContext.WriteStream^.append('>');
lExecuteContext.WriteStream^.newline();

                
END_METHOD

METHOD _reportStateActiveRising
  VAR_INPUT
    state : POINTER TO t_reportablestate;
  END_VAR
                  _reportState(state,FALSE);

                
END_METHOD

METHOD _reportStateUnsuppressFalling
  VAR_INPUT
    state : POINTER TO t_reportablestate;
  END_VAR
                  _reportState(state);


                
END_METHOD

METHOD _reportStateUnsuppressRising
  VAR_INPUT
    state : POINTER TO t_reportablestate;
  END_VAR
                  _reportState(state,FALSE);




                
END_METHOD

PROPERTY VolumeMbs : REAL
GET
                    VolumeMbs := lVolumeMbs;
                  
END_GET
END_PROPERTY

PROPERTY TypeToken : t_medium_string
GET
                    TypeToken := 'RepChanLogTCP';
                  
END_GET
END_PROPERTY

PROPERTY Server : REFERENCE TO TCPServer
GET
                    Server ref= lServer;
                  
END_GET
END_PROPERTY

PROPERTY ChannelConnected : BOOL
GET
                    ChannelConnected := lServer.ClientConnected;

                  
END_GET
END_PROPERTY
END_FUNCTION_BLOCK

FUNCTION_BLOCK EchoTCPServer EXTENDS TCPServer
  VAR
    lHandlers : ARRAY[1..cConnectionsLimit] OF EchoConnectionHandler;
  END_VAR

            
          

METHOD initialize
  VAR
    i : USINT;
  END_VAR
                  FOR i:=1 TO cConnectionsLimit DO
	lConnections[i].Handler := ADR(lHandlers[i]);
END_FOR

SUPER^.initialize();

                
END_METHOD

PROPERTY TypeToken : t_medium_string
GET
                    TypeToken := 'EchoTCPServer';
                  
END_GET
END_PROPERTY
END_FUNCTION_BLOCK

FUNCTION_BLOCK NullTCPServer EXTENDS TCPServer
  VAR
    lHandlers : ARRAY[1..cConnectionsLimit] OF ConnectionHandler;
  END_VAR

            
          

METHOD initialize
  VAR
    i : USINT;
  END_VAR
                  

FOR i:=1 TO cConnectionsLimit DO
	lConnections[i].Handler := ADR(lHandlers[i]);
END_FOR

SUPER^.initialize();

                
END_METHOD

PROPERTY TypeToken : t_medium_string
GET
                    TypeToken := 'TCPServer';
                  
END_GET
END_PROPERTY
END_FUNCTION_BLOCK

FUNCTION_BLOCK ParseTCPServer EXTENDS TCPServer
  VAR
    lHandlers : ARRAY[1..cConnectionsLimit] OF ParseConnectionHandler;
    lReadWrite : BOOL := FALSE;
  END_VAR

            
          

METHOD initialize
  VAR
    i : USINT;
  END_VAR
                  FOR i:=1 TO cConnectionsLimit DO
	lHandlers[i].initialize();
	lConnections[i].Handler := ADR(lHandlers[i]);
	lConnections[i].EnableSkipCompletingNewline := TRUE;
END_FOR

SUPER^.initialize();

                
END_METHOD

PROPERTY WrappedResponse : BOOL
SET
  VAR
    i : USINT;
  END_VAR
                    FOR i:=1 TO cConnectionsLimit DO
	lHandlers[i].ExecuteContext^.WrappedResponse := WrappedResponse;
END_FOR
                  
END_SET
END_PROPERTY

PROPERTY ReportError : BOOL
SET
  VAR
    i : USINT;
  END_VAR
                    FOR i:=1 TO cConnectionsLimit DO
	lHandlers[i].ExecuteContext^.ReportError := ReportError;
END_FOR
                  
END_SET
END_PROPERTY

PROPERTY TypeToken : t_medium_string
GET
                    TypeToken := 'ParseTCPServer';
                  
END_GET
END_PROPERTY

PROPERTY ReadWrite : BOOL
GET
                    ReadWrite := lReadWrite;
                  
END_GET
SET
  VAR
    i : USINT;
  END_VAR
                    lReadWrite := ReadWrite;

FOR i:=1 TO cConnectionsLimit DO
	lHandlers[i].ReadWrite := TRUE;
END_FOR
                  
END_SET
END_PROPERTY

PROPERTY Interactive : BOOL
SET
  VAR
    i : USINT;
  END_VAR
                    FOR i:=1 TO cConnectionsLimit DO
	lHandlers[i].Interactive := Interactive;
END_FOR
                  
END_SET
END_PROPERTY
END_FUNCTION_BLOCK

FUNCTION_BLOCK TCPClient EXTENDS NonOperationalParticleSet
  VAR
    lVRServerPort : ValueReferenceUINT;
    lServerPort : WORD := 49700;
    lAttemptsLimit : USINT := 10;
    lAttempts : USINT;
    lState : t_socket_state;
    lCloseCount : UINT := 0;
    lClientHandle : RTS_IEC_HANDLE;
    lSocketAddress : SOCKADDRESS;
    lSendReturnValue : DINT;
    lSysSockIoCtl_Param : DINT := 1;  (* 1 enabling non-blocking, pdiParameter := 0 disabling non-blocking *)
    lCreateResult : SysTypes.RTS_IEC_RESULT := 1;
    lIOCtlResult : SysTypes.RTS_IEC_RESULT := 1;
    lBindResult : SysTypes.RTS_IEC_RESULT := 1;
    lConnectResult : SysTypes.RTS_IEC_RESULT := 1;
    lSendResult : SysTypes.RTS_IEC_RESULT;
    lCloseResult : SysTypes.RTS_IEC_RESULT := 1;
    lBuffer : ARRAY[0..1400] OF BYTE;
    lWritten : UINT := 0;
  END_VAR

            
          

METHOD close
                  lCloseResult := SysSockClose(hSocket := lClientHandle);
 
IF (lCloseResult=CmpErrors.Errors.ERR_OK) THEN   
	lState := cSocketStateCreate;
END_IF

lClientHandle := SysTypes.RTS_INVALID_HANDLE;
lState := cSocketStateCreate; //foobar

                
END_METHOD

METHOD operator
                  CASE lState OF
	cSocketStateCreate:
		create();
		
	cSocketStateIOCtl:
		ioctl();
		
	cSocketStateBind:
		bind();
		
	cSocketStateConnect:
		connect();
		
	cSocketStateConnected:
		connected();
		
	cSocketStateClose:
		close();
END_CASE

	
                
END_METHOD

METHOD create
                  lClientHandle := SysSockCreate(iAddressFamily := SOCKET_AF_INET,
	diType := SOCKET_STREAM,
	diProtocol := SOCKET_IPPROTO_TCP, 
	pResult := ADR(lCreateResult));
 	
IF ((lClientHandle<>SysTypes.RTS_INVALID_HANDLE) AND
	(lCreateResult=CmpErrors.Errors.ERR_OK)) THEN
	lState := cSocketStateIOCtl;
END_IF
                
END_METHOD

METHOD ioctl
                  lIOCtlResult := SysSockIoctl(hSocket := lClientHandle,
	diCommand := SOCKET_FIONBIO,
	pdiParameter := ADR(lSysSockIoCtl_Param));
	  
IF (lIOCtlResult=CmpErrors.Errors.ERR_OK) THEN   
	lState := cSocketStateConnect;
END_IF
  
                
END_METHOD

METHOD connected
                  ;
                
END_METHOD

METHOD initialize
                  lVRServerPort.initializeValueReference(lServerPort,NopSelf,'Port','Default port','',cValueStyleParameter);

lState := cSocketStateCreate;
lCloseCount := 0;
lAttempts := 0;

lClientHandle := SysTypes.RTS_INVALID_HANDLE;

SUPER^.initialize();
                
END_METHOD

METHOD bind
                  lState := cSocketStateConnect;
                
END_METHOD

METHOD write
  VAR_INPUT
    buffer : POINTER TO BYTE;
    length : UINT;
  END_VAR
                  IF (lState<>cSocketStateConnected) THEN
	operator();
	IF (lState<>cSocketStateConnected) THEN
		RETURN;
	END_IF
END_IF

IF (length=0) THEN
	RETURN;
END_IF

lWritten := lWritten + length;

lSendReturnValue := TO_DINT(SysSockSend(hSocket := lClientHandle,
	pbyBuffer := buffer,
	diBufferSize := length,  
	diFlags := 0,
	pResult := ADR(lSendResult)));
	
IF ((lSendReturnValue<>length) OR
	(lSendResult<>CmpErrors.Errors.ERR_OK)) THEN   
	lState := cSocketStateClose;
	lCloseCount := lCloseCount + 1;
END_IF
                
END_METHOD

METHOD connect
                        // Create a connection from this client to a TCP server
lSocketAddress.sin_family := SOCKET_AF_INET;
lSocketAddress.sin_port := SysSockHtons(usHost := lServerPort);

lSocketAddress.sin_addr.S_un_b.s_b1 := 10;
lSocketAddress.sin_addr.S_un_b.s_b2 := 2; 
lSocketAddress.sin_addr.S_un_b.s_b3 := 3; 
lSocketAddress.sin_addr.S_un_b.s_b4 := 10;

lConnectResult := SysSockConnect(hSocket := lClientHandle,
	pSockAddr := ADR(lSocketAddress),
	diSockAddrSize := SIZEOF(lSocketAddress)); 
 
IF (lConnectResult=CmpErrors.Errors.ERR_OK) THEN   
	lState := cSocketStateConnected;
END_IF

                
END_METHOD

PROPERTY ClientConnected : BOOL
GET
                    ClientConnected := (lState=cSocketStateConnected);

                  
END_GET
END_PROPERTY

PROPERTY ServerPort : WORD
GET
                    ServerPort := lServerPort;
                  
END_GET
SET
                    lServerPort := ServerPort;


                  
END_SET
END_PROPERTY

PROPERTY TypeToken : t_medium_string
GET
                    TypeToken := 'TCPClient';
                  
END_GET
END_PROPERTY
END_FUNCTION_BLOCK

FUNCTION_BLOCK TCPConnection
  VAR
    lState : t_socket_state;
    lServerHandle : RTS_IEC_HANDLE := SysTypes.RTS_INVALID_HANDLE;
    lClientHandle : RTS_IEC_HANDLE := SysTypes.RTS_INVALID_HANDLE;
    lAcceptResult : SysTypes.RTS_IEC_RESULT;
    lIOCtlResult : SysTypes.RTS_IEC_RESULT;
    lSendResult : SysTypes.RTS_IEC_RESULT;
    lRecvResult : SysTypes.RTS_IEC_RESULT;
    lCloseResult : SysTypes.RTS_IEC_RESULT;
    lSocketAddress : SOCKADDRESS;
    lSocketAddressSize : DINT := SIZEOF(lSocketAddress);
    lSysSockIoCtl_Param : DINT := 1;  (* 1 enabling non-blocking, pdiParameter := 0 disabling non-blocking *)
    lSendReturnValue : DINT;
    lRecvReturnValue : DINT;
    lSuppressRead : BOOL := FALSE;
    lSuppressWrite : BOOL := FALSE;
    lOverflowError : UINT := 0;
    lWriteError : UINT := 0;
    lReadError : UINT := 0;
    lHandler : POINTER TO t_connection_handler := 0;
    lConnectionCount : UINT := 0;
    lReadCount : UINT := 0;
    lWriteCount : UINT := 0;
    lEnableSkipCompletingNewline : BOOL := FALSE;
    lSkipCompletingNewline : BOOL := FALSE;
    lSkipInitialMessages : USINT := 0;
  END_VAR

            
          

METHOD write
  VAR_INPUT
    buffer : POINTER TO BYTE;
    length : UINT;
  END_VAR
                  IF (lState<>cSocketStateConnected) THEN
	RETURN;
END_IF

IF (length=0) THEN
	RETURN;
END_IF

IF (lSuppressWrite) THEN
	RETURN;
END_IF

lSendReturnValue := TO_DINT(SysSockSend(hSocket := lClientHandle,
	pbyBuffer := buffer,
	diBufferSize := length,  
	diFlags := 0,
	pResult := ADR(lSendResult)));

IF (lSendResult=CmpErrors.Errors.ERR_OK) THEN
	lWriteCount := lWriteCount + 1;
	RETURN;
END_IF

IF (lSendResult=CmpErrors.Errors.ERR_SOCK_CLOSED) THEN
	lState := cSocketStateClose;

	RETURN;
END_IF

IF ((lSendReturnValue<>length) OR
	(lSendResult=CmpErrors.Errors.ERR_SOCK_WOULDBLOCK)) THEN  
	lOverflowError := lOverflowError + 1;
	lState := cSocketStateClose;

	RETURN;
END_IF

lWriteError := lWriteError + 1;
lState := cSocketStateClose;

                
END_METHOD

METHOD close
                  lCloseResult := SysSockClose(hSocket := lClientHandle);

lClientHandle := SysTypes.RTS_INVALID_HANDLE;
lState := cSocketStateInvalid;



                
END_METHOD

METHOD initialize
                  lState := cSocketStateInvalid;
lConnectionCount := 0;

lServerHandle := SysTypes.RTS_INVALID_HANDLE;
lClientHandle := SysTypes.RTS_INVALID_HANDLE;
                
END_METHOD

METHOD operator
                  CASE lState OF
	cSocketStateInvalid:
		invalid();
		
	cSocketStateConnect:
		connect();
		
	cSocketStateIOCtl:
		ioctl();

	cSocketStateConnected:
		connected();
		
	cSocketStateClose:
		close();
END_CASE

	
                
END_METHOD

METHOD connect
                  IF (NOT(fIsValidTCPHandle(lServerHandle))) THEN
	lState := cSocketStateInvalid;
	RETURN;
END_IF
  
lClientHandle := SysSockAccept(hSocket := lServerHandle,
	pSockAddr := ADR(lSocketAddress), 
	pdiSockAddrSize := ADR(lSocketAddressSize),
	pResult := ADR(lAcceptResult));

IF (fIsValidTCPHandle(lClientHandle)) THEN
	lState := cSocketStateIOCtl;
	lConnectionCount := lConnectionCount + 1;
END_IF
                
END_METHOD

METHOD connected
                  IF (lHandler=0) THEN
	RETURN;
END_IF

lHandler^.operator();

                
END_METHOD

METHOD invalid
                  IF (fIsValidTCPHandle(lServerHandle)) THEN
	lState := cSocketStateConnect;
END_IF
                
END_METHOD

METHOD read : BOOL
  VAR_INPUT
    stream : POINTER TO t_stream;
  END_VAR
  VAR
    buffer : POINTER TO BYTE;
  END_VAR
                  IF (lState<>cSocketStateConnected) THEN
	read := FALSE;
	RETURN;
END_IF

IF (stream=0) THEN
	read := FALSE;
	RETURN;
END_IF

IF (SuppressRead) THEN
	read := FALSE;
	RETURN;
END_IF

IF (NOT(fIsValidTCPHandle(lClientHandle))) THEN
	read := FALSE;
	RETURN;
END_IF

lRecvReturnValue := TO_DINT(SysSockRecv(hSocket := lClientHandle,
	pbyBuffer := stream^.Buffer,
	diBufferSize := stream^.cBufferUseableSize,
	diFlags := 0,
	pResult := ADR(lRecvResult)));

IF (lRecvReturnValue>0) THEN
	stream^.Length := TO_UINT(lRecvReturnValue);
	lReadCount := lReadCount + 1;

	IF (lSkipInitialMessages>0) THEN
		lSkipInitialMessages := lSkipInitialMessages - 1;
		read := FALSE;
		RETURN;
	END_IF

	IF (lEnableSkipCompletingNewline) THEN
		buffer := stream^.Buffer;

		read := NOT((lSkipCompletingNewline) AND
			(lRecvReturnValue=2) AND 
			(buffer[0]=13) AND
			(buffer[1]=10));
		
		lSkipCompletingNewline := (lRecvReturnValue>2);
	ELSE
		read := TRUE;
	END_IF	
		
	RETURN;
END_IF

IF ((lRecvResult=CmpErrors.Errors.ERR_OK) OR
	(lRecvResult=CmpErrors.Errors.ERR_SOCK_WOULDBLOCK)) THEN
	read := FALSE;
	RETURN;
END_IF

IF (lRecvResult=CmpErrors.Errors.ERR_SOCK_CLOSED) THEN
	lState := cSocketStateClose;

	read := FALSE;
	RETURN;
END_IF

lReadError := lReadError + 1;
lState := cSocketStateClose;
read := FALSE;


                
END_METHOD

METHOD ioctl
                  lIOCtlResult := SysSockIoctl(hSocket := lClientHandle,
	diCommand := SOCKET_FIONBIO,
	pdiParameter := ADR(lSysSockIoCtl_Param));

IF (lIOCtlResult=CmpErrors.Errors.ERR_OK) THEN   	
	lSkipCompletingNewline := FALSE;
	lState := cSocketStateConnected;

	IF (lHandler<>0) THEN
		lHandler^.connecting();
		RETURN;
	END_IF
END_IF

                
END_METHOD

PROPERTY ServerHandle : RTS_IEC_HANDLE
GET
                    ServerHandle := lServerHandle;
                  
END_GET
SET
                    lServerHandle := ServerHandle;

                  
END_SET
END_PROPERTY

PROPERTY SuppressRead : BOOL
GET
                    SuppressRead := lSuppressRead;
                  
END_GET
SET
                    lSuppressRead := SuppressRead;
                  
END_SET
END_PROPERTY

PROPERTY SuppressWrite : BOOL
GET
                    SuppressWrite := lSuppressWrite;
                  
END_GET
SET
                    lSuppressWrite := SuppressWrite;
                  
END_SET
END_PROPERTY

PROPERTY Handler : POINTER TO t_connection_handler
GET
                    Handler := lHandler;
                  
END_GET
SET
                    lHandler := Handler;

IF (lHandler<>0) THEN
	lHandler^.Connection := THIS;
END_IF
                  
END_SET
END_PROPERTY

PROPERTY EnableSkipCompletingNewline : BOOL
GET
                    EnableSkipCompletingNewline := lEnableSkipCompletingNewline;
                  
END_GET
SET
                    lEnableSkipCompletingNewline := EnableSkipCompletingNewline;
                  
END_SET
END_PROPERTY

PROPERTY SkipInitialMessages : USINT
GET
                    SkipInitialMessages := lSkipInitialMessages;
                  
END_GET
SET
                    lSkipInitialMessages := SkipInitialMessages;
                  
END_SET
END_PROPERTY

PROPERTY ClientConnected : BOOL
GET
                    ClientConnected := (lState=cSocketStateConnected);

                  
END_GET
END_PROPERTY
END_FUNCTION_BLOCK

FUNCTION_BLOCK TCPServer EXTENDS NonOperationalParticleSet
  VAR CONSTANT
    cConnectionsLimit : USINT := 2;
  END_VAR
  VAR
    lVRServerPort : ValueReferenceUINT;
    lServerPort : UINT := 49860;
    lVRServerPortLower : ValueReferenceUINT;
    lServerPortLower : UINT := 49860;
    lVRServerPortUpper : ValueReferenceUINT;
    lServerPortUpper : UINT := 49869;
    lEnabled : BOOL := TRUE;
    lSuppressWrite : BOOL := FALSE;
    lAttemptsLimit : USINT := 10;
    lAttempts : USINT;
    lCurrentServerPort : WORD;
    lState : t_socket_state;
    lConnectionCount : UINT := 0;
    lServerHandle : RTS_IEC_HANDLE;
    lSocketAddress : SOCKADDRESS;
    lSysSockIoCtl_Param : DINT := 1;  (* 1 enabling non-blocking, pdiParameter := 0 disabling non-blocking *)
    lCreateResult : SysTypes.RTS_IEC_RESULT;
    lIOCtlResult : SysTypes.RTS_IEC_RESULT;
    lBindResult : SysTypes.RTS_IEC_RESULT;
    lListenResult : SysTypes.RTS_IEC_RESULT;
    lCloseResult : SysTypes.RTS_IEC_RESULT;
    lConnections : ARRAY[1..cConnectionsLimit] OF t_tcp_connection;
    lClientConnected : BOOL := FALSE;
  END_VAR

            
          

METHOD create
                  lServerHandle := SysSockCreate(iAddressFamily := SOCKET_AF_INET,
	diType := SOCKET_STREAM,
	diProtocol := SOCKET_IPPROTO_TCP, 
	pResult := ADR(lCreateResult));
	
IF ((fIsValidTCPHandle(lServerHandle)) AND
	(lCreateResult=CmpErrors.Errors.ERR_OK)) THEN
	lState := cSocketStateIOCtl;
	
	lConnectionCount := lConnectionCount + 1;
END_IF

                
END_METHOD

METHOD initialize
                  lVRServerPortLower.initializeValueReference(lServerPortLower,NopSelf,'PortLower','Lower end of port range','',cValueStyleParameter);
lVRServerPortUpper.initializeValueReference(lServerPortUpper,NopSelf,'PortUpper','Upper end of port range','',cValueStyleParameter);
lVRServerPort.initializeValueReference(lServerPort,NopSelf,'Port','Default port','',cValueStyleParameter);

lState := cSocketStateCreate;
lConnectionCount := 0;

lCurrentServerPort := lServerPort;
lAttempts := 0;

lServerHandle := SysTypes.RTS_INVALID_HANDLE;

SUPER^.initialize();

                
END_METHOD

METHOD write
  VAR_INPUT
    buffer : POINTER TO BYTE;
    length : UINT;
  END_VAR
  VAR
    i : USINT;
  END_VAR
                  IF (lState<>cSocketStateConnect) THEN
	RETURN;
END_IF

IF (length=0) THEN
	RETURN;
END_IF

IF (lSuppressWrite) THEN
	RETURN;
END_IF

FOR i:=1 TO cConnectionsLimit DO
	lConnections[i].write(buffer,length);
END_FOR

                
END_METHOD

METHOD close
  VAR
    i : USINT;
  END_VAR
                  lCloseResult := SysSockClose(hSocket := lServerHandle);
 
lCurrentServerPort := lServerPort;
lAttempts := 0;

lServerHandle := SysTypes.RTS_INVALID_HANDLE;
lState := cSocketStateCreate;

FOR i:=1 TO cConnectionsLimit DO
	lConnections[i].close();
	lConnections[i].ServerHandle := lServerHandle;
END_FOR

                
END_METHOD

METHOD ioctl
                  lIOCtlResult := SysSockIoctl(hSocket := lServerHandle,
	diCommand := SOCKET_FIONBIO,
	pdiParameter := ADR(lSysSockIoCtl_Param));
	  
IF (lIOCtlResult=CmpErrors.Errors.ERR_OK) THEN   
	lState := cSocketStateBind;
END_IF
	  

                
END_METHOD

METHOD operator
  VAR
    i : USINT;
  END_VAR
                  IF (NOT(lEnabled)) THEN
	RETURN;
END_IF

CASE lState OF
	cSocketStateCreate:
		create();
		
	cSocketStateIOCtl:
		ioctl();
		
	cSocketStateBind:
		bind();
		
	cSocketStateListen:
		listen();
		
	cSocketStateConnect:
		connect();
		
	cSocketStateClose:
		close();
END_CASE

lClientConnected := FALSE;
FOR i:=1 TO cConnectionsLimit DO
	lConnections[i].operator();
	IF (lConnections[i].ClientConnected) THEN
		lClientConnected := TRUE;
	END_IF
END_FOR

	
                
END_METHOD

METHOD bind
                  IF ((lCurrentServerPort<lServerPortLower) OR
	(lCurrentServerPort>lServerPortUpper)) THEN
	lCurrentServerPort := lServerPortLower;
END_IF

lSocketAddress.sin_family := SOCKET_AF_INET;
lSocketAddress.sin_port := SysSockHtons(usHost := lCurrentServerPort);    
lSocketAddress.sin_addr.ulAddr := SOCKET_INADDR_ANY;

lBindResult := SysSockBind(hSocket := lServerHandle,
	pSockAddr := ADR(lSocketAddress),
	diSockAddrSize := SIZEOF(lSocketAddress));
 
IF (lBindResult=CmpErrors.Errors.ERR_OK) THEN 
	lState := cSocketStateListen;
ELSE
	lAttempts := lAttempts + 1;
	
	IF (lAttempts>=lAttemptsLimit) THEN
		lAttempts := 0;
	
		lCurrentServerPort := lCurrentServerPort + 1;
		IF (lCurrentServerPort>lServerPortUpper) THEN
			lCurrentServerPort := lServerPortLower;
		END_IF
	END_IF
END_IF

                
END_METHOD

METHOD connect
                  ;

                
END_METHOD

METHOD listen
  VAR
    i : USINT;
  END_VAR
                  lListenResult := SysSockListen(hSocket := lServerHandle,
	diMaxConnections := cConnectionsLimit); 
 
IF (lListenResult=CmpErrors.Errors.ERR_OK) THEN   
	lState := cSocketStateConnect;
	
	FOR i:=1 TO cConnectionsLimit DO
		lConnections[i].ServerHandle := lServerHandle;
	END_FOR
//ELSE
	//lState := cSocketStateClose;
END_IF

                
END_METHOD

METHOD execute
  VAR_INPUT
    executeContext : POINTER TO ExecuteContext;
  END_VAR
                  IF (executeContext^.matchCommand(sCommandClose)) THEN	
	close();
	RETURN;
END_IF

SUPER^.execute(executeContext);

                
END_METHOD

METHOD describe
  VAR_INPUT
    executeContext : POINTER TO ExecuteContext;
  END_VAR
                  SUPER^.describe(executeContext);

IF (executeContext^.matchOption(cExecuteOptionSyntax)) THEN
	executeContext^.describeSyntaxExecutable(sCommandClose);
	RETURN;
END_IF


                
END_METHOD

PROPERTY ServerPort : UINT
GET
                    ServerPort := lServerPort;
                  
END_GET
SET
                    lServerPort := ServerPort;
lCurrentServerPort := lServerPort;

                  
END_SET
END_PROPERTY

PROPERTY Enabled : BOOL
GET
                    Enabled := lEnabled;

                  
END_GET
SET
                    lEnabled := Enabled;
                  
END_SET
END_PROPERTY

PROPERTY SuppressWrite : BOOL
GET
                    SuppressWrite := lSuppressWrite;
                  
END_GET
SET
                    lSuppressWrite := SuppressWrite;
                  
END_SET
END_PROPERTY

PROPERTY TypeToken : t_medium_string
GET
                    TypeToken := 'TCPServer';
                  
END_GET
END_PROPERTY

PROPERTY ServerPortLower : UINT
GET
                    ServerPortLower := lServerPortLower;
                  
END_GET
SET
                    lServerPortLower := ServerPortLower;


                  
END_SET
END_PROPERTY

PROPERTY ServerPortUpper : UINT
GET
                    ServerPortUpper := lServerPortUpper;
                  
END_GET
SET
                    lServerPortUpper := ServerPortUpper;


                  
END_SET
END_PROPERTY

PROPERTY ClientConnected : BOOL
GET
                    ClientConnected := lClientConnected;
                  
END_GET
END_PROPERTY
END_FUNCTION_BLOCK

